LIN {X 0,Y 310.79,Z 469.746,A -85,B 0,C 180,E1 -15567.408,E2 -15567.408} C_VEL
LIN {X 0,Y 310.865,Z 470.154,A -85,B 0,C 180,E1 -15568.705,E2 -15568.705} C_VEL
LIN {X 0,Y 311.02,Z 469.974,A -85,B 0,C 180,E1 -15570,E2 -15570} C_VEL
LIN {X 0,Y 310.921,Z 469.285,A -85,B 0,C 180,E1 -15571.296,E2 -15571.296} C_VEL
LIN {X 0,Y 310.834,Z 468.094,A -85,B 0,C 180,E1 -15572.592,E2 -15572.592} C_VEL
LIN {X 0,Y 310.902,Z 466.384,A -85,B 0,C 180,E1 -15573.889,E2 -15573.889} C_VEL
LIN {X 0,Y 310.831,Z 464.037,A -85,B 0,C 180,E1 -15575.189,E2 -15575.189} C_VEL
LIN {X 0,Y 311.032,Z 459.255,A -85,B 0,C 180,E1 -15577.139,E2 -15577.139} C_VEL
LIN {X 0,Y 311.34,Z 454.023,A -85,B 0,C 180,E1 -15578.764,E2 -15578.764} C_VEL
LIN {X 0,Y 311.659,Z 448.881,A -85,B 0,C 180,E1 -15580.065,E2 -15580.065} C_VEL
LIN {X 0,Y 312.198,Z 442.687,A -85,B 0,C 180,E1 -15581.36,E2 -15581.36} C_VEL
LIN {X 0,Y 312.796,Z 436.181,A -85,B 0,C 180,E1 -15582.489,E2 -15582.489} C_VEL
LIN {X 0,Y 313.49,Z 428.304,A -85,B 0,C 180,E1 -15583.615,E2 -15583.615} C_VEL
LIN {X 0,Y 314.177,Z 420.016,A -85,B 0,C 180,E1 -15584.576,E2 -15584.576} C_VEL
LIN {X 0,Y 314.912,Z 409.522,A -85,B 0,C 180,E1 -15585.534,E2 -15585.534} C_VEL
LIN {X 0,Y 315.686,Z 397.677,A -85,B 0,C 180,E1 -15586.282,E2 -15586.282} C_VEL
LIN {X 0,Y 316.118,Z 388.576,A -85,B 0,C 180,E1 -15586.674,E2 -15586.674} C_VEL
LIN {X 0,Y 316.81,Z 345.999,A -85,B 0,C 180,E1 -15587.795,E2 -15587.795} C_VEL
LIN {X 0,Y 313.032,Z 310.136,A -85,B 0,C 180,E1 -15588.921,E2 -15588.921} C_VEL
LIN {X 0,Y 314.417,Z 295.649,A -85,B 0,C 180,E1 -15593.027,E2 -15593.027} C_VEL
LIN {X 0,Y 314.951,Z 289.674,A -85,B 0,C 180,E1 -15594.733,E2 -15594.733} C_VEL
LIN {X 0,Y 313.279,Z 279.811,A -85,B 0,C 180,E1 -15597.742,E2 -15597.742} C_VEL
LIN {X 0,Y 312.618,Z 276.356,A -85,B 0,C 180,E1 -15598.878,E2 -15598.878} C_VEL
LIN {X 0,Y 312.505,Z 276.368,A -85,B 0,C 180,E1 -15602.666,E2 -15602.666} C_VEL
LIN {X 0,Y 312.538,Z 276.365,A -85,B 0,C 180,E1 -15605.949,E2 -15605.949} C_VEL
LIN {X 0,Y 312.509,Z 276.368,A -85,B 0,C 180,E1 -15609.027,E2 -15609.027} C_VEL
LIN {X 0,Y 312.513,Z 276.366,A -85,B 0,C 180,E1 -15612.427,E2 -15612.427} C_VEL
LIN {X 0,Y 312.458,Z 276.375,A -85,B 0,C 180,E1 -15616.034,E2 -15616.034} C_VEL
LIN {X 0,Y 312.504,Z 276.37,A -85,B 0,C 180,E1 -15619.874,E2 -15619.874} C_VEL
LIN {X 0,Y 312.534,Z 276.365,A -85,B 0,C 180,E1 -15624.05,E2 -15624.05} C_VEL
LIN {X 0,Y 312.504,Z 276.371,A -85,B 0,C 180,E1 -15627.333,E2 -15627.333} C_VEL
LIN {X 0,Y 312.551,Z 276.364,A -85,B 0,C 180,E1 -15631.275,E2 -15631.275} C_VEL
LIN {X 0,Y 312.584,Z 276.358,A -85,B 0,C 180,E1 -15634.71,E2 -15634.71} C_VEL
LIN {X 0,Y 312.585,Z 276.362,A -85,B 0,C 180,E1 -15637.528,E2 -15637.528} C_VEL
LIN {X 0,Y 312.636,Z 276.356,A -85,B 0,C 180,E1 -15641.655,E2 -15641.655} C_VEL
LIN {X 0,Y 312.691,Z 276.349,A -85,B 0,C 180,E1 -15645.685,E2 -15645.685} C_VEL
LIN {X 0,Y 312.695,Z 276.349,A -85,B 0,C 180,E1 -15649.641,E2 -15649.641} C_VEL
LIN {X 0,Y 312.85,Z 276.325,A -85,B 0,C 180,E1 -15652.253,E2 -15652.253} C_VEL
LIN {X 0,Y 312.712,Z 276.341,A -85,B 0,C 180,E1 -15654.841,E2 -15654.841} C_VEL
LIN {X 0,Y 312.986,Z 276.307,A -85,B 0,C 180,E1 -15658.712,E2 -15658.712} C_VEL
LIN {X 0,Y 312.986,Z 276.31,A -85,B 0,C 180,E1 -15661.286,E2 -15661.286} C_VEL
LIN {X 0,Y 312.713,Z 276.343,A -85,B 0,C 180,E1 -15665.157,E2 -15665.157} C_VEL
LIN {X 0,Y 312.867,Z 276.327,A -85,B 0,C 180,E1 -15667.745,E2 -15667.745} C_VEL
LIN {X 0,Y 312.666,Z 276.353,A -85,B 0,C 180,E1 -15671.67,E2 -15671.67} C_VEL
LIN {X 0,Y 312.694,Z 276.344,A -85,B 0,C 180,E1 -15674.886,E2 -15674.886} C_VEL
LIN {X 0,Y 312.627,Z 276.354,A -85,B 0,C 180,E1 -15679.237,E2 -15679.237} C_VEL
LIN {X 0,Y 312.54,Z 276.363,A -85,B 0,C 180,E1 -15682.788,E2 -15682.788} C_VEL
LIN {X 0,Y 312.596,Z 276.359,A -85,B 0,C 180,E1 -15685.934,E2 -15685.934} C_VEL
LIN {X 0,Y 312.538,Z 276.368,A -85,B 0,C 180,E1 -15689.649,E2 -15689.649} C_VEL
LIN {X 0,Y 312.512,Z 276.372,A -85,B 0,C 180,E1 -15693.688,E2 -15693.688} C_VEL
LIN {X 0,Y 312.545,Z 276.365,A -85,B 0,C 180,E1 -15697.381,E2 -15697.381} C_VEL
LIN {X 0,Y 312.495,Z 276.369,A -85,B 0,C 180,E1 -15700.706,E2 -15700.706} C_VEL
LIN {X 0,Y 312.524,Z 276.366,A -85,B 0,C 180,E1 -15704.195,E2 -15704.195} C_VEL
LIN {X 0,Y 312.542,Z 276.367,A -85,B 0,C 180,E1 -15707.905,E2 -15707.905} C_VEL
LIN {X 0,Y 312.55,Z 276.366,A -85,B 0,C 180,E1 -15711.904,E2 -15711.904} C_VEL
LIN {X 0,Y 312.498,Z 276.374,A -85,B 0,C 180,E1 -15715.789,E2 -15715.789} C_VEL
LIN {X 0,Y 312.515,Z 276.366,A -85,B 0,C 180,E1 -15718.853,E2 -15718.853} C_VEL
LIN {X 0,Y 312.566,Z 276.365,A -85,B 0,C 180,E1 -15721.824,E2 -15721.824} C_VEL
LIN {X 0,Y 312.577,Z 276.358,A -85,B 0,C 180,E1 -15724.71,E2 -15724.71} C_VEL
LIN {X 0,Y 312.579,Z 276.361,A -85,B 0,C 180,E1 -15727.529,E2 -15727.529} C_VEL
LIN {X 0,Y 312.63,Z 276.356,A -85,B 0,C 180,E1 -15731.656,E2 -15731.656} C_VEL
LIN {X 0,Y 312.686,Z 276.35,A -85,B 0,C 180,E1 -15735.686,E2 -15735.686} C_VEL
LIN {X 0,Y 312.694,Z 276.348,A -85,B 0,C 180,E1 -15739.641,E2 -15739.641} C_VEL
LIN {X 0,Y 312.863,Z 276.324,A -85,B 0,C 180,E1 -15742.254,E2 -15742.254} C_VEL
LIN {X 0,Y 312.707,Z 276.342,A -85,B 0,C 180,E1 -15744.842,E2 -15744.842} C_VEL
LIN {X 0,Y 312.982,Z 276.308,A -85,B 0,C 180,E1 -15748.713,E2 -15748.713} C_VEL
LIN {X 0,Y 312.982,Z 276.309,A -85,B 0,C 180,E1 -15751.286,E2 -15751.286} C_VEL
LIN {X 0,Y 312.705,Z 276.343,A -85,B 0,C 180,E1 -15755.157,E2 -15755.157} C_VEL
LIN {X 0,Y 312.857,Z 276.328,A -85,B 0,C 180,E1 -15757.746,E2 -15757.746} C_VEL
LIN {X 0,Y 312.663,Z 276.352,A -85,B 0,C 180,E1 -15761.671,E2 -15761.671} C_VEL
LIN {X 0,Y 312.691,Z 276.344,A -85,B 0,C 180,E1 -15764.887,E2 -15764.887} C_VEL
LIN {X 0,Y 312.62,Z 276.354,A -85,B 0,C 180,E1 -15769.236,E2 -15769.236} C_VEL
LIN {X 0,Y 312.518,Z 276.366,A -85,B 0,C 180,E1 -15772.781,E2 -15772.781} C_VEL
LIN {X 0,Y 312.592,Z 276.362,A -85,B 0,C 180,E1 -15775.935,E2 -15775.935} C_VEL
LIN {X 0,Y 312.628,Z 276.487,A -85,B 0,C 180,E1 -15780.151,E2 -15780.151} C_VEL
LIN {X 0,Y 316.262,Z 290.124,A -85,B 0,C 180,E1 -15780.69,E2 -15780.69} C_VEL
LIN {X 0,Y 317.61,Z 298.066,A -85,B 0,C 180,E1 -15780.961,E2 -15780.961} C_VEL
LIN {X 0,Y 316.407,Z 353.531,A -85,B 0,C 180,E1 -15782.395,E2 -15782.395} C_VEL
LIN {X 0,Y 316.063,Z 363.172,A -85,B 0,C 180,E1 -15782.81,E2 -15782.81} C_VEL
LIN {X 0,Y 315.661,Z 373.664,A -85,B 0,C 180,E1 -15783.469,E2 -15783.469} C_VEL
LIN {X 0,Y 315.027,Z 383.974,A -85,B 0,C 180,E1 -15784.37,E2 -15784.37} C_VEL
LIN {X 0,Y 314.498,Z 392.833,A -85,B 0,C 180,E1 -15785.373,E2 -15785.373} C_VEL
LIN {X 0,Y 313.829,Z 400.58,A -85,B 0,C 180,E1 -15786.45,E2 -15786.45} C_VEL
LIN {X 0,Y 313.237,Z 406.85,A -85,B 0,C 180,E1 -15787.496,E2 -15787.496} C_VEL
LIN {X 0,Y 312.678,Z 413.25,A -85,B 0,C 180,E1 -15788.781,E2 -15788.781} C_VEL
LIN {X 0,Y 312.251,Z 418.582,A -85,B 0,C 180,E1 -15790.073,E2 -15790.073} C_VEL
LIN {X 0,Y 311.761,Z 423.009,A -85,B 0,C 180,E1 -15791.357,E2 -15791.357} C_VEL
LIN {X 0,Y 311.393,Z 427.97,A -85,B 0,C 180,E1 -15793.173,E2 -15793.173} C_VEL
LIN {X 0,Y 311.139,Z 430.66,A -85,B 0,C 180,E1 -15794.444,E2 -15794.444} C_VEL
LIN {X 0,Y 310.846,Z 433.632,A -85,B 0,C 180,E1 -15796.342,E2 -15796.342} C_VEL
LIN {X 0,Y 310.717,Z 435.486,A -85,B 0,C 180,E1 -15798.279,E2 -15798.279} C_VEL
LIN {X 0,Y 310.853,Z 436.168,A -85,B 0,C 180,E1 -15800.235,E2 -15800.235} C_VEL
LIN {X 0,Y 311.126,Z 435.457,A -85,B 0,C 180,E1 -15802.42,E2 -15802.42} C_VEL
LIN {X 0,Y 311.755,Z 432.834,A -85,B 0,C 180,E1 -15805.016,E2 -15805.016} C_VEL
LIN {X 0,Y 312.419,Z 429.501,A -85,B 0,C 180,E1 -15806.874,E2 -15806.874} C_VEL
LIN {X 0,Y 313.123,Z 425.447,A -85,B 0,C 180,E1 -15808.526,E2 -15808.526} C_VEL
LIN {X 0,Y 313.952,Z 420.392,A -85,B 0,C 180,E1 -15810.129,E2 -15810.129} C_VEL
LIN {X 0,Y 314.722,Z 415.473,A -85,B 0,C 180,E1 -15811.397,E2 -15811.397} C_VEL
LIN {X 0,Y 315.617,Z 410.145,A -85,B 0,C 180,E1 -15812.541,E2 -15812.541} C_VEL
LIN {X 0,Y 316.642,Z 402.89,A -85,B 0,C 180,E1 -15813.825,E2 -15813.825} C_VEL
LIN {X 0,Y 316.901,Z 401.141,A -85,B 0,C 180,E1 -15814.099,E2 -15814.099} C_VEL
LIN {X 0,Y 316.944,Z 396.688,A -85,B 0,C 180,E1 -15814.803,E2 -15814.803} C_VEL
LIN {X 0,Y 315.234,Z 389.246,A -85,B 0,C 180,E1 -15815.954,E2 -15815.954} C_VEL
LIN {X 0,Y 313.375,Z 381.279,A -85,B 0,C 180,E1 -15816.97,E2 -15816.97} C_VEL
LIN {X 0,Y 313.161,Z 376.007,A -85,B 0,C 180,E1 -15817.451,E2 -15817.451} C_VEL
LIN {X 0,Y 313.835,Z 365.078,A -85,B 0,C 180,E1 -15818.166,E2 -15818.166} C_VEL
LIN {X 0,Y 314.322,Z 354.986,A -85,B 0,C 180,E1 -15818.61,E2 -15818.61} C_VEL
LIN {X 0,Y 315.93,Z 301.668,A -85,B 0,C 180,E1 -15820.067,E2 -15820.067} C_VEL
LIN {X 0,Y 309.852,Z 287.044,A -85,B 0,C 180,E1 -15821.116,E2 -15821.116} C_VEL
LIN {X 0,Y 305.843,Z 278.339,A -85,B 0,C 180,E1 -15821.842,E2 -15821.842} C_VEL
LIN {X 0,Y 305.572,Z 277.239,A -85,B 0,C 180,E1 -15822.259,E2 -15822.259} C_VEL
LIN {X 0,Y 305.64,Z 277.227,A -85,B 0,C 180,E1 -15825.35,E2 -15825.35} C_VEL
LIN {X 0,Y 305.627,Z 277.228,A -85,B 0,C 180,E1 -15829.401,E2 -15829.401} C_VEL
LIN {X 0,Y 305.789,Z 277.206,A -85,B 0,C 180,E1 -15832.075,E2 -15832.075} C_VEL
LIN {X 0,Y 305.682,Z 277.217,A -85,B 0,C 180,E1 -15834.725,E2 -15834.725} C_VEL
LIN {X 0,Y 305.95,Z 277.186,A -85,B 0,C 180,E1 -15838.685,E2 -15838.685} C_VEL
LIN {X 0,Y 305.952,Z 277.181,A -85,B 0,C 180,E1 -15841.317,E2 -15841.317} C_VEL
LIN {X 0,Y 305.845,Z 277.201,A -85,B 0,C 180,E1 -15846.599,E2 -15846.599} C_VEL
LIN {X 0,Y 305.729,Z 277.211,A -85,B 0,C 180,E1 -15849.261,E2 -15849.261} C_VEL
LIN {X 0,Y 305.582,Z 277.228,A -85,B 0,C 180,E1 -15853.297,E2 -15853.297} C_VEL
LIN {X 0,Y 305.588,Z 277.225,A -85,B 0,C 180,E1 -15856.021,E2 -15856.021} C_VEL
LIN {X 0,Y 305.572,Z 277.231,A -85,B 0,C 180,E1 -15859.446,E2 -15859.446} C_VEL
LIN {X 0,Y 305.485,Z 277.243,A -85,B 0,C 180,E1 -15863.042,E2 -15863.042} C_VEL
LIN {X 0,Y 305.549,Z 277.23,A -85,B 0,C 180,E1 -15866.231,E2 -15866.231} C_VEL
LIN {X 0,Y 305.491,Z 277.234,A -85,B 0,C 180,E1 -15869.051,E2 -15869.051} C_VEL
LIN {X 0,Y 305.441,Z 277.251,A -85,B 0,C 180,E1 -15871.953,E2 -15871.953} C_VEL
LIN {X 0,Y 305.459,Z 277.249,A -85,B 0,C 180,E1 -15875.115,E2 -15875.115} C_VEL
LIN {X 0,Y 305.48,Z 277.245,A -85,B 0,C 180,E1 -15878.538,E2 -15878.538} C_VEL
LIN {X 0,Y 305.494,Z 277.245,A -85,B 0,C 180,E1 -15882.595,E2 -15882.595} C_VEL
LIN {X 0,Y 305.442,Z 277.248,A -85,B 0,C 180,E1 -15886.349,E2 -15886.349} C_VEL
LIN {X 0,Y 305.457,Z 277.249,A -85,B 0,C 180,E1 -15889.894,E2 -15889.894} C_VEL
LIN {X 0,Y 305.499,Z 277.244,A -85,B 0,C 180,E1 -15893.628,E2 -15893.628} C_VEL
LIN {X 0,Y 305.465,Z 277.248,A -85,B 0,C 180,E1 -15896.484,E2 -15896.484} C_VEL
LIN {X 0,Y 305.472,Z 277.401,A -85,B 0,C 180,E1 -15898.423,E2 -15898.423} C_VEL
LIN {X 0,Y 307.594,Z 285.931,A -85,B 0,C 180,E1 -15901.328,E2 -15901.328} C_VEL
LIN {X 0,Y 309.242,Z 294.45,A -85,B 0,C 180,E1 -15904.057,E2 -15904.057} C_VEL
LIN {X 0,Y 309.221,Z 297.943,A -85,B 0,C 180,E1 -15905.076,E2 -15905.076} C_VEL
LIN {X 0,Y 308.121,Z 306.513,A -85,B 0,C 180,E1 -15907.455,E2 -15907.455} C_VEL
LIN {X 0,Y 311.702,Z 324.802,A -85,B 0,C 180,E1 -15908.395,E2 -15908.395} C_VEL
LIN {X 0,Y 314.275,Z 342.889,A -85,B 0,C 180,E1 -15909.166,E2 -15909.166} C_VEL
LIN {X 0,Y 314.794,Z 351.131,A -85,B 0,C 180,E1 -15909.452,E2 -15909.452} C_VEL
LIN {X 0,Y 313.562,Z 387.051,A -85,B 0,C 180,E1 -15910.439,E2 -15910.439} C_VEL
LIN {X 0,Y 312.761,Z 399.292,A -85,B 0,C 180,E1 -15911.02,E2 -15911.02} C_VEL
LIN {X 0,Y 311.652,Z 409.779,A -85,B 0,C 180,E1 -15911.767,E2 -15911.767} C_VEL
LIN {X 0,Y 310.591,Z 418.26,A -85,B 0,C 180,E1 -15912.554,E2 -15912.554} C_VEL
LIN {X 0,Y 309.461,Z 426.47,A -85,B 0,C 180,E1 -15913.509,E2 -15913.509} C_VEL
LIN {X 0,Y 308.325,Z 434.313,A -85,B 0,C 180,E1 -15914.635,E2 -15914.635} C_VEL
LIN {X 0,Y 307.201,Z 440.849,A -85,B 0,C 180,E1 -15915.764,E2 -15915.764} C_VEL
LIN {X 0,Y 306.261,Z 447.117,A -85,B 0,C 180,E1 -15917.072,E2 -15917.072} C_VEL
LIN {X 0,Y 305.279,Z 453.551,A -85,B 0,C 180,E1 -15918.716,E2 -15918.716} C_VEL
LIN {X 0,Y 304.439,Z 459.551,A -85,B 0,C 180,E1 -15920.701,E2 -15920.701} C_VEL
LIN {X 0,Y 304.07,Z 462.704,A -85,B 0,C 180,E1 -15922.029,E2 -15922.029} C_VEL
LIN {X 0,Y 303.732,Z 466.505,A -85,B 0,C 180,E1 -15924.255,E2 -15924.255} C_VEL
LIN {X 0,Y 303.723,Z 468.469,A -85,B 0,C 180,E1 -15926.02,E2 -15926.02} C_VEL
LIN {X 0,Y 303.71,Z 469.371,A -85,B 0,C 180,E1 -15927.348,E2 -15927.348} C_VEL
LIN {X 0,Y 303.77,Z 469.762,A -85,B 0,C 180,E1 -15928.675,E2 -15928.675} C_VEL
LIN {X 0,Y 303.93,Z 469.549,A -85,B 0,C 180,E1 -15930,E2 -15930} C_VEL
LIN {X 0,Y 303.828,Z 468.81,A -85,B 0,C 180,E1 -15931.326,E2 -15931.326} C_VEL
LIN {X 0,Y 303.755,Z 467.568,A -85,B 0,C 180,E1 -15932.653,E2 -15932.653} C_VEL
LIN {X 0,Y 303.832,Z 465.805,A -85,B 0,C 180,E1 -15933.979,E2 -15933.979} C_VEL
LIN {X 0,Y 303.812,Z 462.107,A -85,B 0,C 180,E1 -15935.893,E2 -15935.893} C_VEL
LIN {X 0,Y 303.961,Z 458.545,A -85,B 0,C 180,E1 -15937.306,E2 -15937.306} C_VEL
LIN {X 0,Y 304.281,Z 453.238,A -85,B 0,C 180,E1 -15938.969,E2 -15938.969} C_VEL
LIN {X 0,Y 304.647,Z 448.017,A -85,B 0,C 180,E1 -15940.299,E2 -15940.299} C_VEL
LIN {X 0,Y 305.185,Z 441.723,A -85,B 0,C 180,E1 -15941.625,E2 -15941.625} C_VEL
LIN {X 0,Y 305.816,Z 435.104,A -85,B 0,C 180,E1 -15942.779,E2 -15942.779} C_VEL
LIN {X 0,Y 306.489,Z 427.078,A -85,B 0,C 180,E1 -15943.932,E2 -15943.932} C_VEL
LIN {X 0,Y 307.377,Z 417.101,A -85,B 0,C 180,E1 -15945.075,E2 -15945.075} C_VEL
LIN {X 0,Y 308.176,Z 406.544,A -85,B 0,C 180,E1 -15945.967,E2 -15945.967} C_VEL
LIN {X 0,Y 308.774,Z 396.77,A -85,B 0,C 180,E1 -15946.572,E2 -15946.572} C_VEL
LIN {X 0,Y 309.194,Z 387.415,A -85,B 0,C 180,E1 -15946.974,E2 -15946.974} C_VEL
LIN {X 0,Y 309.893,Z 346.657,A -85,B 0,C 180,E1 -15948.07,E2 -15948.07} C_VEL
LIN {X 0,Y 306.062,Z 309.72,A -85,B 0,C 180,E1 -15949.263,E2 -15949.263} C_VEL
LIN {X 0,Y 307.516,Z 295.348,A -85,B 0,C 180,E1 -15953.44,E2 -15953.44} C_VEL
LIN {X 0,Y 307.887,Z 290.114,A -85,B 0,C 180,E1 -15954.979,E2 -15954.979} C_VEL
LIN {X 0,Y 306.129,Z 280.199,A -85,B 0,C 180,E1 -15958.075,E2 -15958.075} C_VEL
LIN {X 0,Y 305.557,Z 277.236,A -85,B 0,C 180,E1 -15959.069,E2 -15959.069} C_VEL
LIN {X 0,Y 305.467,Z 277.25,A -85,B 0,C 180,E1 -15963.516,E2 -15963.516} C_VEL
LIN {X 0,Y 305.482,Z 277.242,A -85,B 0,C 180,E1 -15966.738,E2 -15966.738} C_VEL
LIN {X 0,Y 305.456,Z 277.245,A -85,B 0,C 180,E1 -15970.599,E2 -15970.599} C_VEL
LIN {X 0,Y 305.429,Z 277.253,A -85,B 0,C 180,E1 -15973.654,E2 -15973.654} C_VEL
LIN {X 0,Y 305.455,Z 277.25,A -85,B 0,C 180,E1 -15977.413,E2 -15977.413} C_VEL
LIN {X 0,Y 305.475,Z 277.248,A -85,B 0,C 180,E1 -15981.597,E2 -15981.597} C_VEL
LIN {X 0,Y 305.461,Z 277.245,A -85,B 0,C 180,E1 -15984.886,E2 -15984.886} C_VEL
LIN {X 0,Y 305.451,Z 277.246,A -85,B 0,C 180,E1 -15988.354,E2 -15988.354} C_VEL
LIN {X 0,Y 305.519,Z 277.239,A -85,B 0,C 180,E1 -15991.113,E2 -15991.113} C_VEL
LIN {X 0,Y 305.57,Z 277.233,A -85,B 0,C 180,E1 -15994.087,E2 -15994.087} C_VEL
LIN {X 0,Y 305.498,Z 277.24,A -85,B 0,C 180,E1 -15998.402,E2 -15998.402} C_VEL
LIN {X 0,Y 305.588,Z 277.231,A -85,B 0,C 180,E1 -16001.217,E2 -16001.217} C_VEL
LIN {X 0,Y 305.646,Z 277.225,A -85,B 0,C 180,E1 -16005.348,E2 -16005.348} C_VEL
LIN {X 0,Y 305.632,Z 277.227,A -85,B 0,C 180,E1 -16009.398,E2 -16009.398} C_VEL
LIN {X 0,Y 305.794,Z 277.205,A -85,B 0,C 180,E1 -16012.073,E2 -16012.073} C_VEL
LIN {X 0,Y 305.683,Z 277.217,A -85,B 0,C 180,E1 -16014.722,E2 -16014.722} C_VEL
LIN {X 0,Y 305.953,Z 277.184,A -85,B 0,C 180,E1 -16018.683,E2 -16018.683} C_VEL
LIN {X 0,Y 305.953,Z 277.186,A -85,B 0,C 180,E1 -16021.315,E2 -16021.315} C_VEL
LIN {X 0,Y 305.847,Z 277.197,A -85,B 0,C 180,E1 -16026.596,E2 -16026.596} C_VEL
LIN {X 0,Y 305.731,Z 277.213,A -85,B 0,C 180,E1 -16029.259,E2 -16029.259} C_VEL
LIN {X 0,Y 305.585,Z 277.231,A -85,B 0,C 180,E1 -16033.295,E2 -16033.295} C_VEL
LIN {X 0,Y 305.588,Z 277.231,A -85,B 0,C 180,E1 -16036.019,E2 -16036.019} C_VEL
LIN {X 0,Y 305.575,Z 277.234,A -85,B 0,C 180,E1 -16039.446,E2 -16039.446} C_VEL
LIN {X 0,Y 305.484,Z 277.242,A -85,B 0,C 180,E1 -16043.04,E2 -16043.04} C_VEL
LIN {X 0,Y 305.525,Z 277.238,A -85,B 0,C 180,E1 -16046.22,E2 -16046.22} C_VEL
LIN {X 0,Y 305.487,Z 277.242,A -85,B 0,C 180,E1 -16049.048,E2 -16049.048} C_VEL
LIN {X 0,Y 305.437,Z 277.251,A -85,B 0,C 180,E1 -16051.951,E2 -16051.951} C_VEL
LIN {X 0,Y 305.456,Z 277.246,A -85,B 0,C 180,E1 -16055.112,E2 -16055.112} C_VEL
LIN {X 0,Y 305.484,Z 277.242,A -85,B 0,C 180,E1 -16058.538,E2 -16058.538} C_VEL
LIN {X 0,Y 305.491,Z 277.241,A -85,B 0,C 180,E1 -16062.594,E2 -16062.594} C_VEL
LIN {X 0,Y 305.489,Z 277.242,A -85,B 0,C 180,E1 -16066.357,E2 -16066.357} C_VEL
LIN {X 0,Y 305.477,Z 277.247,A -85,B 0,C 180,E1 -16069.896,E2 -16069.896} C_VEL
LIN {X 0,Y 305.494,Z 277.245,A -85,B 0,C 180,E1 -16073.626,E2 -16073.626} C_VEL
LIN {X 0,Y 305.457,Z 277.246,A -85,B 0,C 180,E1 -16076.483,E2 -16076.483} C_VEL
LIN {X 0,Y 305.487,Z 277.242,A -85,B 0,C 180,E1 -16080.95,E2 -16080.95} C_VEL
LIN {X 0,Y 305.563,Z 277.234,A -85,B 0,C 180,E1 -16084.087,E2 -16084.087} C_VEL
LIN {X 0,Y 305.493,Z 277.242,A -85,B 0,C 180,E1 -16088.402,E2 -16088.402} C_VEL
LIN {X 0,Y 305.582,Z 277.23,A -85,B 0,C 180,E1 -16091.217,E2 -16091.217} C_VEL
LIN {X 0,Y 305.641,Z 277.224,A -85,B 0,C 180,E1 -16095.349,E2 -16095.349} C_VEL
LIN {X 0,Y 305.63,Z 277.226,A -85,B 0,C 180,E1 -16099.399,E2 -16099.399} C_VEL
LIN {X 0,Y 305.804,Z 277.205,A -85,B 0,C 180,E1 -16102.074,E2 -16102.074} C_VEL
LIN {X 0,Y 305.679,Z 277.218,A -85,B 0,C 180,E1 -16104.723,E2 -16104.723} C_VEL
LIN {X 0,Y 305.948,Z 277.184,A -85,B 0,C 180,E1 -16108.683,E2 -16108.683} C_VEL
LIN {X 0,Y 305.948,Z 277.185,A -85,B 0,C 180,E1 -16111.316,E2 -16111.316} C_VEL
LIN {X 0,Y 305.837,Z 277.198,A -85,B 0,C 180,E1 -16116.597,E2 -16116.597} C_VEL
LIN {X 0,Y 305.727,Z 277.212,A -85,B 0,C 180,E1 -16119.259,E2 -16119.259} C_VEL
LIN {X 0,Y 305.582,Z 277.231,A -85,B 0,C 180,E1 -16123.296,E2 -16123.296} C_VEL
LIN {X 0,Y 305.585,Z 277.233,A -85,B 0,C 180,E1 -16126.02,E2 -16126.02} C_VEL
LIN {X 0,Y 305.566,Z 277.234,A -85,B 0,C 180,E1 -16129.444,E2 -16129.444} C_VEL
LIN {X 0,Y 305.477,Z 277.243,A -85,B 0,C 180,E1 -16133.039,E2 -16133.039} C_VEL
LIN {X 0,Y 305.522,Z 277.24,A -85,B 0,C 180,E1 -16136.221,E2 -16136.221} C_VEL
LIN {X 0,Y 305.565,Z 277.237,A -85,B 0,C 180,E1 -16139.791,E2 -16139.791} C_VEL
LIN {X 0,Y 309.356,Z 290.796,A -85,B 0,C 180,E1 -16140.382,E2 -16140.382} C_VEL
LIN {X 0,Y 310.704,Z 298.29,A -85,B 0,C 180,E1 -16140.647,E2 -16140.647} C_VEL
LIN {X 0,Y 309.438,Z 354.306,A -85,B 0,C 180,E1 -16142.137,E2 -16142.137} C_VEL
LIN {X 0,Y 309.141,Z 365.224,A -85,B 0,C 180,E1 -16142.639,E2 -16142.639} C_VEL
LIN {X 0,Y 308.53,Z 376.572,A -85,B 0,C 180,E1 -16143.432,E2 -16143.432} C_VEL
LIN {X 0,Y 307.94,Z 385.711,A -85,B 0,C 180,E1 -16144.292,E2 -16144.292} C_VEL
LIN {X 0,Y 307.458,Z 393.812,A -85,B 0,C 180,E1 -16145.251,E2 -16145.251} C_VEL
LIN {X 0,Y 306.774,Z 401.469,A -85,B 0,C 180,E1 -16146.353,E2 -16146.353} C_VEL
LIN {X 0,Y 306.028,Z 409.075,A -85,B 0,C 180,E1 -16147.692,E2 -16147.692} C_VEL
LIN {X 0,Y 305.364,Z 416.54,A -85,B 0,C 180,E1 -16149.323,E2 -16149.323} C_VEL
LIN {X 0,Y 304.707,Z 423.154,A -85,B 0,C 180,E1 -16151.21,E2 -16151.21} C_VEL
LIN {X 0,Y 304.446,Z 426.533,A -85,B 0,C 180,E1 -16152.381,E2 -16152.381} C_VEL
LIN {X 0,Y 304.089,Z 430.667,A -85,B 0,C 180,E1 -16154.239,E2 -16154.239} C_VEL
LIN {X 0,Y 303.785,Z 433.584,A -85,B 0,C 180,E1 -16156.051,E2 -16156.051} C_VEL
LIN {X 0,Y 303.63,Z 435.461,A -85,B 0,C 180,E1 -16157.838,E2 -16157.838} C_VEL
LIN {X 0,Y 303.716,Z 436.438,A -85,B 0,C 180,E1 -16159.783,E2 -16159.783} C_VEL
LIN {X 0,Y 303.918,Z 436.314,A -85,B 0,C 180,E1 -16161.833,E2 -16161.833} C_VEL
LIN {X 0,Y 304.376,Z 434.864,A -85,B 0,C 180,E1 -16163.913,E2 -16163.913} C_VEL
LIN {X 0,Y 305.156,Z 431.279,A -85,B 0,C 180,E1 -16166.446,E2 -16166.446} C_VEL
LIN {X 0,Y 306.11,Z 426.596,A -85,B 0,C 180,E1 -16168.595,E2 -16168.595} C_VEL
LIN {X 0,Y 307.057,Z 421.034,A -85,B 0,C 180,E1 -16170.427,E2 -16170.427} C_VEL
LIN {X 0,Y 307.866,Z 416.322,A -85,B 0,C 180,E1 -16171.689,E2 -16171.689} C_VEL
LIN {X 0,Y 309.043,Z 409.67,A -85,B 0,C 180,E1 -16173.131,E2 -16173.131} C_VEL
LIN {X 0,Y 310.193,Z 401.975,A -85,B 0,C 180,E1 -16174.487,E2 -16174.487} C_VEL
LIN {X 0,Y 311.326,Z 393.583,A -85,B 0,C 180,E1 -16175.679,E2 -16175.679} C_VEL
LIN {X 0,Y 312.472,Z 382.935,A -85,B 0,C 180,E1 -16176.854,E2 -16176.854} C_VEL
LIN {X 0,Y 313.161,Z 376.007,A -85,B 0,C 180,E1 -16177.451,E2 -16177.451} C_VEL
LIN {X 0,Y 313.02,Z 370.58,A -85,B 0,C 180,E1 -16177.886,E2 -16177.886} C_VEL
LIN {X 0,Y 310.949,Z 361.716,A -85,B 0,C 180,E1 -16178.611,E2 -16178.611} C_VEL
LIN {X 0,Y 308.672,Z 352.653,A -85,B 0,C 180,E1 -16179.206,E2 -16179.206} C_VEL
LIN {X 0,Y 308.201,Z 346.919,A -85,B 0,C 180,E1 -16179.434,E2 -16179.434} C_VEL
LIN {X 0,Y 309.684,Z 303.662,A -85,B 0,C 180,E1 -16180.617,E2 -16180.617} C_VEL
LIN {X 0,Y 303.269,Z 288.312,A -85,B 0,C 180,E1 -16181.771,E2 -16181.771} C_VEL
LIN {X 0,Y 299.412,Z 280.754,A -85,B 0,C 180,E1 -16182.455,E2 -16182.455} C_VEL
LIN {X 0,Y 298.668,Z 278.879,A -85,B 0,C 180,E1 -16182.631,E2 -16182.631} C_VEL
LIN {X 0,Y 298.529,Z 278.114,A -85,B 0,C 180,E1 -16182.975,E2 -16182.975} C_VEL
LIN {X 0,Y 298.543,Z 278.11,A -85,B 0,C 180,E1 -16186.386,E2 -16186.386} C_VEL
LIN {X 0,Y 298.72,Z 278.09,A -85,B 0,C 180,E1 -16191.156,E2 -16191.156} C_VEL
LIN {X 0,Y 298.781,Z 278.082,A -85,B 0,C 180,E1 -16193.247,E2 -16193.247} C_VEL
LIN {X 0,Y 298.916,Z 278.061,A -85,B 0,C 180,E1 -16198.654,E2 -16198.654} C_VEL
LIN {X 0,Y 298.918,Z 278.057,A -85,B 0,C 180,E1 -16201.348,E2 -16201.348} C_VEL
LIN {X 0,Y 298.791,Z 278.078,A -85,B 0,C 180,E1 -16206.755,E2 -16206.755} C_VEL
LIN {X 0,Y 298.674,Z 278.091,A -85,B 0,C 180,E1 -16209.482,E2 -16209.482} C_VEL
LIN {X 0,Y 298.546,Z 278.106,A -85,B 0,C 180,E1 -16213.617,E2 -16213.617} C_VEL
LIN {X 0,Y 298.543,Z 278.1,A -85,B 0,C 180,E1 -16216.41,E2 -16216.41} C_VEL
LIN {X 0,Y 298.507,Z 278.111,A -85,B 0,C 180,E1 -16219.656,E2 -16219.656} C_VEL
LIN {X 0,Y 298.453,Z 278.118,A -85,B 0,C 180,E1 -16223.599,E2 -16223.599} C_VEL
LIN {X 0,Y 298.488,Z 278.113,A -85,B 0,C 180,E1 -16226.576,E2 -16226.576} C_VEL
LIN {X 0,Y 298.417,Z 278.114,A -85,B 0,C 180,E1 -16229.642,E2 -16229.642} C_VEL
LIN {X 0,Y 298.392,Z 278.121,A -85,B 0,C 180,E1 -16232.802,E2 -16232.802} C_VEL
LIN {X 0,Y 298.463,Z 278.113,A -85,B 0,C 180,E1 -16236.814,E2 -16236.814} C_VEL
LIN {X 0,Y 298.417,Z 278.121,A -85,B 0,C 180,E1 -16241.096,E2 -16241.096} C_VEL
LIN {X 0,Y 298.387,Z 278.131,A -85,B 0,C 180,E1 -16244.96,E2 -16244.96} C_VEL
LIN {X 0,Y 298.386,Z 278.127,A -85,B 0,C 180,E1 -16248.914,E2 -16248.914} C_VEL
LIN {X 0,Y 298.426,Z 278.128,A -85,B 0,C 180,E1 -16252.245,E2 -16252.245} C_VEL
LIN {X 0,Y 298.408,Z 278.128,A -85,B 0,C 180,E1 -16255.582,E2 -16255.582} C_VEL
LIN {X 0,Y 298.426,Z 278.287,A -85,B 0,C 180,E1 -16257.77,E2 -16257.77} C_VEL
LIN {X 0,Y 300.702,Z 287.389,A -85,B 0,C 180,E1 -16260.991,E2 -16260.991} C_VEL
LIN {X 0,Y 302.356,Z 295.878,A -85,B 0,C 180,E1 -16263.793,E2 -16263.793} C_VEL
LIN {X 0,Y 302.532,Z 298.325,A -85,B 0,C 180,E1 -16264.549,E2 -16264.549} C_VEL
LIN {X 0,Y 301.482,Z 306.03,A -85,B 0,C 180,E1 -16266.746,E2 -16266.746} C_VEL
LIN {X 0,Y 305.448,Z 326.004,A -85,B 0,C 180,E1 -16267.814,E2 -16267.814} C_VEL
LIN {X 0,Y 307.985,Z 344.653,A -85,B 0,C 180,E1 -16268.643,E2 -16268.643} C_VEL
LIN {X 0,Y 308.373,Z 351.988,A -85,B 0,C 180,E1 -16268.902,E2 -16268.902} C_VEL
LIN {X 0,Y 307.188,Z 386.272,A -85,B 0,C 180,E1 -16269.868,E2 -16269.868} C_VEL
LIN {X 0,Y 306.345,Z 398.258,A -85,B 0,C 180,E1 -16270.428,E2 -16270.428} C_VEL
LIN {X 0,Y 305.157,Z 408.946,A -85,B 0,C 180,E1 -16271.191,E2 -16271.191} C_VEL
LIN {X 0,Y 304.061,Z 417.502,A -85,B 0,C 180,E1 -16271.993,E2 -16271.993} C_VEL
LIN {X 0,Y 302.9,Z 425.769,A -85,B 0,C 180,E1 -16272.967,E2 -16272.967} C_VEL
LIN {X 0,Y 301.814,Z 432.633,A -85,B 0,C 180,E1 -16273.948,E2 -16273.948} C_VEL
LIN {X 0,Y 300.671,Z 439.364,A -85,B 0,C 180,E1 -16275.102,E2 -16275.102} C_VEL
LIN {X 0,Y 299.536,Z 445.789,A -85,B 0,C 180,E1 -16276.431,E2 -16276.431} C_VEL
LIN {X 0,Y 298.715,Z 451.15,A -85,B 0,C 180,E1 -16277.776,E2 -16277.776} C_VEL
LIN {X 0,Y 297.95,Z 455.644,A -85,B 0,C 180,E1 -16279.123,E2 -16279.123} C_VEL
LIN {X 0,Y 297.212,Z 460.997,A -85,B 0,C 180,E1 -16281.159,E2 -16281.159} C_VEL
LIN {X 0,Y 296.763,Z 464.973,A -85,B 0,C 180,E1 -16283.2,E2 -16283.2} C_VEL
LIN {X 0,Y 296.622,Z 466.815,A -85,B 0,C 180,E1 -16284.562,E2 -16284.562} C_VEL
LIN {X 0,Y 296.634,Z 468.151,A -85,B 0,C 180,E1 -16285.925,E2 -16285.925} C_VEL
LIN {X 0,Y 296.631,Z 468.997,A -85,B 0,C 180,E1 -16287.284,E2 -16287.284} C_VEL
LIN {X 0,Y 296.678,Z 469.356,A -85,B 0,C 180,E1 -16288.643,E2 -16288.643} C_VEL
LIN {X 0,Y 296.84,Z 469.12,A -85,B 0,C 180,E1 -16290,E2 -16290} C_VEL
LIN {X 0,Y 296.736,Z 468.321,A -85,B 0,C 180,E1 -16291.357,E2 -16291.357} C_VEL
LIN {X 0,Y 296.678,Z 467.018,A -85,B 0,C 180,E1 -16292.716,E2 -16292.716} C_VEL
LIN {X 0,Y 296.717,Z 464.023,A -85,B 0,C 180,E1 -16294.756,E2 -16294.756} C_VEL
LIN {X 0,Y 296.843,Z 459.683,A -85,B 0,C 180,E1 -16296.799,E2 -16296.799} C_VEL
LIN {X 0,Y 297.177,Z 453.599,A -85,B 0,C 180,E1 -16298.843,E2 -16298.843} C_VEL
LIN {X 0,Y 297.498,Z 448.527,A -85,B 0,C 180,E1 -16300.206,E2 -16300.206} C_VEL
LIN {X 0,Y 298.054,Z 442.416,A -85,B 0,C 180,E1 -16301.562,E2 -16301.562} C_VEL
LIN {X 0,Y 298.765,Z 434.975,A -85,B 0,C 180,E1 -16302.913,E2 -16302.913} C_VEL
LIN {X 0,Y 299.453,Z 427.001,A -85,B 0,C 180,E1 -16304.093,E2 -16304.093} C_VEL
LIN {X 0,Y 300.167,Z 418.6,A -85,B 0,C 180,E1 -16305.098,E2 -16305.098} C_VEL
LIN {X 0,Y 301.079,Z 407.91,A -85,B 0,C 180,E1 -16306.093,E2 -16306.093} C_VEL
LIN {X 0,Y 301.846,Z 396.427,A -85,B 0,C 180,E1 -16306.833,E2 -16306.833} C_VEL
LIN {X 0,Y 302.248,Z 387.103,A -85,B 0,C 180,E1 -16307.246,E2 -16307.246} C_VEL
LIN {X 0,Y 303.038,Z 347.743,A -85,B 0,C 180,E1 -16308.332,E2 -16308.332} C_VEL
LIN {X 0,Y 299.076,Z 309.407,A -85,B 0,C 180,E1 -16309.594,E2 -16309.594} C_VEL
LIN {X 0,Y 300.613,Z 295.01,A -85,B 0,C 180,E1 -16313.873,E2 -16313.873} C_VEL
LIN {X 0,Y 300.773,Z 290.486,A -85,B 0,C 180,E1 -16315.241,E2 -16315.241} C_VEL
LIN {X 0,Y 298.739,Z 279.321,A -85,B 0,C 180,E1 -16318.834,E2 -16318.834} C_VEL
LIN {X 0,Y 298.499,Z 278.117,A -85,B 0,C 180,E1 -16319.274,E2 -16319.274} C_VEL
LIN {X 0,Y 298.397,Z 278.126,A -85,B 0,C 180,E1 -16322.8,E2 -16322.8} C_VEL
LIN {X 0,Y 298.453,Z 278.118,A -85,B 0,C 180,E1 -16326.808,E2 -16326.808} C_VEL
LIN {X 0,Y 298.413,Z 278.124,A -85,B 0,C 180,E1 -16331.092,E2 -16331.092} C_VEL
LIN {X 0,Y 298.355,Z 278.131,A -85,B 0,C 180,E1 -16335.034,E2 -16335.034} C_VEL
LIN {X 0,Y 298.384,Z 278.127,A -85,B 0,C 180,E1 -16338.737,E2 -16338.737} C_VEL
LIN {X 0,Y 298.413,Z 278.123,A -85,B 0,C 180,E1 -16342.241,E2 -16342.241} C_VEL
LIN {X 0,Y 298.408,Z 278.129,A -85,B 0,C 180,E1 -16345.58,E2 -16345.58} C_VEL
LIN {X 0,Y 298.395,Z 278.125,A -85,B 0,C 180,E1 -16348.79,E2 -16348.79} C_VEL
LIN {X 0,Y 298.462,Z 278.119,A -85,B 0,C 180,E1 -16351.903,E2 -16351.903} C_VEL
LIN {X 0,Y 298.484,Z 278.115,A -85,B 0,C 180,E1 -16354.923,E2 -16354.923} C_VEL
LIN {X 0,Y 298.448,Z 278.12,A -85,B 0,C 180,E1 -16359.314,E2 -16359.314} C_VEL
LIN {X 0,Y 298.535,Z 278.109,A -85,B 0,C 180,E1 -16362.178,E2 -16362.178} C_VEL
LIN {X 0,Y 298.591,Z 278.101,A -85,B 0,C 180,E1 -16364.994,E2 -16364.994} C_VEL
LIN {X 0,Y 298.588,Z 278.102,A -85,B 0,C 180,E1 -16369.145,E2 -16369.145} C_VEL
LIN {X 0,Y 298.738,Z 278.085,A -85,B 0,C 180,E1 -16371.884,E2 -16371.884} C_VEL
LIN {X 0,Y 298.654,Z 278.092,A -85,B 0,C 180,E1 -16374.598,E2 -16374.598} C_VEL
LIN {X 0,Y 298.919,Z 278.06,A -85,B 0,C 180,E1 -16378.652,E2 -16378.652} C_VEL
LIN {X 0,Y 298.919,Z 278.063,A -85,B 0,C 180,E1 -16381.346,E2 -16381.346} C_VEL
LIN {X 0,Y 298.793,Z 278.076,A -85,B 0,C 180,E1 -16386.753,E2 -16386.753} C_VEL
LIN {X 0,Y 298.676,Z 278.094,A -85,B 0,C 180,E1 -16389.479,E2 -16389.479} C_VEL
LIN {X 0,Y 298.548,Z 278.11,A -85,B 0,C 180,E1 -16393.614,E2 -16393.614} C_VEL
LIN {X 0,Y 298.543,Z 278.107,A -85,B 0,C 180,E1 -16396.408,E2 -16396.408} C_VEL
LIN {X 0,Y 298.51,Z 278.116,A -85,B 0,C 180,E1 -16399.656,E2 -16399.656} C_VEL
LIN {X 0,Y 298.451,Z 278.122,A -85,B 0,C 180,E1 -16403.597,E2 -16403.597} C_VEL
LIN {X 0,Y 298.48,Z 278.114,A -85,B 0,C 180,E1 -16406.574,E2 -16406.574} C_VEL
LIN {X 0,Y 298.413,Z 278.127,A -85,B 0,C 180,E1 -16409.64,E2 -16409.64} C_VEL
LIN {X 0,Y 298.389,Z 278.126,A -85,B 0,C 180,E1 -16412.799,E2 -16412.799} C_VEL
LIN {X 0,Y 298.463,Z 278.116,A -85,B 0,C 180,E1 -16416.813,E2 -16416.813} C_VEL
LIN {X 0,Y 298.412,Z 278.124,A -85,B 0,C 180,E1 -16421.094,E2 -16421.094} C_VEL
LIN {X 0,Y 298.452,Z 278.119,A -85,B 0,C 180,E1 -16423.115,E2 -16423.115} C_VEL
LIN {X 0,Y 298.46,Z 278.116,A -85,B 0,C 180,E1 -16426.932,E2 -16426.932} C_VEL
LIN {X 0,Y 298.429,Z 278.121,A -85,B 0,C 180,E1 -16430.998,E2 -16430.998} C_VEL
LIN {X 0,Y 298.426,Z 278.124,A -85,B 0,C 180,E1 -16433.932,E2 -16433.932} C_VEL
LIN {X 0,Y 298.387,Z 278.129,A -85,B 0,C 180,E1 -16437.983,E2 -16437.983} C_VEL
LIN {X 0,Y 298.455,Z 278.121,A -85,B 0,C 180,E1 -16441.904,E2 -16441.904} C_VEL
LIN {X 0,Y 298.478,Z 278.115,A -85,B 0,C 180,E1 -16444.924,E2 -16444.924} C_VEL
LIN {X 0,Y 298.442,Z 278.121,A -85,B 0,C 180,E1 -16449.315,E2 -16449.315} C_VEL
LIN {X 0,Y 298.53,Z 278.11,A -85,B 0,C 180,E1 -16452.179,E2 -16452.179} C_VEL
LIN {X 0,Y 298.585,Z 278.102,A -85,B 0,C 180,E1 -16454.994,E2 -16454.994} C_VEL
LIN {X 0,Y 298.586,Z 278.102,A -85,B 0,C 180,E1 -16459.146,E2 -16459.146} C_VEL
LIN {X 0,Y 298.75,Z 278.085,A -85,B 0,C 180,E1 -16461.886,E2 -16461.886} C_VEL
LIN {X 0,Y 298.65,Z 278.094,A -85,B 0,C 180,E1 -16464.599,E2 -16464.599} C_VEL
LIN {X 0,Y 298.915,Z 278.06,A -85,B 0,C 180,E1 -16468.652,E2 -16468.652} C_VEL
LIN {X 0,Y 298.915,Z 278.062,A -85,B 0,C 180,E1 -16471.347,E2 -16471.347} C_VEL
LIN {X 0,Y 298.783,Z 278.076,A -85,B 0,C 180,E1 -16476.754,E2 -16476.754} C_VEL
LIN {X 0,Y 298.672,Z 278.093,A -85,B 0,C 180,E1 -16479.48,E2 -16479.48} C_VEL
LIN {X 0,Y 298.544,Z 278.11,A -85,B 0,C 180,E1 -16483.615,E2 -16483.615} C_VEL
LIN {X 0,Y 298.54,Z 278.108,A -85,B 0,C 180,E1 -16486.408,E2 -16486.408} C_VEL
LIN {X 0,Y 298.501,Z 278.115,A -85,B 0,C 180,E1 -16489.654,E2 -16489.654} C_VEL
LIN {X 0,Y 298.419,Z 278.125,A -85,B 0,C 180,E1 -16493.6,E2 -16493.6} C_VEL
LIN {X 0,Y 298.478,Z 278.116,A -85,B 0,C 180,E1 -16496.575,E2 -16496.575} C_VEL
LIN {X 0,Y 298.528,Z 278.131,A -85,B 0,C 180,E1 -16499.499,E2 -16499.499} C_VEL
LIN {X 0,Y 302.575,Z 292.277,A -85,B 0,C 180,E1 -16500.103,E2 -16500.103} C_VEL
LIN {X 0,Y 303.818,Z 299.911,A -85,B 0,C 180,E1 -16500.374,E2 -16500.374} C_VEL
LIN {X 0,Y 302.506,Z 354.653,A -85,B 0,C 180,E1 -16501.867,E2 -16501.867} C_VEL
LIN {X 0,Y 302.191,Z 366.027,A -85,B 0,C 180,E1 -16502.405,E2 -16502.405} C_VEL
LIN {X 0,Y 301.587,Z 376.783,A -85,B 0,C 180,E1 -16503.178,E2 -16503.178} C_VEL
LIN {X 0,Y 300.953,Z 386.213,A -85,B 0,C 180,E1 -16504.086,E2 -16504.086} C_VEL
LIN {X 0,Y 300.4,Z 394.895,A -85,B 0,C 180,E1 -16505.147,E2 -16505.147} C_VEL
LIN {X 0,Y 299.765,Z 401.644,A -85,B 0,C 180,E1 -16506.146,E2 -16506.146} C_VEL
LIN {X 0,Y 299.105,Z 408.193,A -85,B 0,C 180,E1 -16507.304,E2 -16507.304} C_VEL
LIN {X 0,Y 298.535,Z 414.281,A -85,B 0,C 180,E1 -16508.597,E2 -16508.597} C_VEL
LIN {X 0,Y 298.103,Z 419.273,A -85,B 0,C 180,E1 -16509.864,E2 -16509.864} C_VEL
LIN {X 0,Y 297.57,Z 424.271,A -85,B 0,C 180,E1 -16511.398,E2 -16511.398} C_VEL
LIN {X 0,Y 297.258,Z 428.142,A -85,B 0,C 180,E1 -16512.87,E2 -16512.87} C_VEL
LIN {X 0,Y 296.904,Z 431.97,A -85,B 0,C 180,E1 -16514.757,E2 -16514.757} C_VEL
LIN {X 0,Y 296.618,Z 434.617,A -85,B 0,C 180,E1 -16516.6,E2 -16516.6} C_VEL
LIN {X 0,Y 296.538,Z 436.252,A -85,B 0,C 180,E1 -16518.427,E2 -16518.427} C_VEL
LIN {X 0,Y 296.665,Z 436.94,A -85,B 0,C 180,E1 -16520.238,E2 -16520.238} C_VEL
LIN {X 0,Y 296.86,Z 436.725,A -85,B 0,C 180,E1 -16522.011,E2 -16522.011} C_VEL
LIN {X 0,Y 297.254,Z 435.639,A -85,B 0,C 180,E1 -16523.768,E2 -16523.768} C_VEL
LIN {X 0,Y 297.82,Z 433.452,A -85,B 0,C 180,E1 -16525.681,E2 -16525.681} C_VEL
LIN {X 0,Y 298.4,Z 430.911,A -85,B 0,C 180,E1 -16527.202,E2 -16527.202} C_VEL
LIN {X 0,Y 299.197,Z 427.173,A -85,B 0,C 180,E1 -16528.886,E2 -16528.886} C_VEL
LIN {X 0,Y 300.074,Z 422.426,A -85,B 0,C 180,E1 -16530.54,E2 -16530.54} C_VEL
LIN {X 0,Y 301.155,Z 416.454,A -85,B 0,C 180,E1 -16532.179,E2 -16532.179} C_VEL
LIN {X 0,Y 302.392,Z 409.932,A -85,B 0,C 180,E1 -16533.611,E2 -16533.611} C_VEL
LIN {X 0,Y 303.467,Z 403.025,A -85,B 0,C 180,E1 -16534.861,E2 -16534.861} C_VEL
LIN {X 0,Y 304.444,Z 396.423,A -85,B 0,C 180,E1 -16535.848,E2 -16535.848} C_VEL
LIN {X 0,Y 305.517,Z 387.505,A -85,B 0,C 180,E1 -16536.944,E2 -16536.944} C_VEL
LIN {X 0,Y 306.68,Z 376.705,A -85,B 0,C 180,E1 -16537.962,E2 -16537.962} C_VEL
LIN {X 0,Y 307.428,Z 365.215,A -85,B 0,C 180,E1 -16538.727,E2 -16538.727} C_VEL
LIN {X 0,Y 307.922,Z 355.353,A -85,B 0,C 180,E1 -16539.17,E2 -16539.17} C_VEL
LIN {X 0,Y 308.201,Z 346.919,A -85,B 0,C 180,E1 -16539.434,E2 -16539.434} C_VEL
LIN {X 0,Y 307.779,Z 341.138,A -85,B 0,C 180,E1 -16539.651,E2 -16539.651} C_VEL
LIN {X 0,Y 303.361,Z 322.574,A -85,B 0,C 180,E1 -16540.669,E2 -16540.669} C_VEL
LIN {X 0,Y 303.017,Z 316.793,A -85,B 0,C 180,E1 -16540.888,E2 -16540.888} C_VEL
LIN {X 0,Y 303.411,Z 305.521,A -85,B 0,C 180,E1 -16541.206,E2 -16541.206} C_VEL
LIN {X 0,Y 296.952,Z 290.192,A -85,B 0,C 180,E1 -16542.425,E2 -16542.425} C_VEL
LIN {X 0,Y 292.827,Z 282.311,A -85,B 0,C 180,E1 -16543.19,E2 -16543.19} C_VEL
LIN {X 0,Y 291.667,Z 279.919,A -85,B 0,C 180,E1 -16543.419,E2 -16543.419} C_VEL
LIN {X 0,Y 291.534,Z 279.215,A -85,B 0,C 180,E1 -16543.547,E2 -16543.547} C_VEL
LIN {X 0,Y 291.495,Z 278.99,A -85,B 0,C 180,E1 -16543.904,E2 -16543.904} C_VEL
LIN {X 0,Y 291.512,Z 278.986,A -85,B 0,C 180,E1 -16547.47,E2 -16547.47} C_VEL
LIN {X 0,Y 291.68,Z 278.965,A -85,B 0,C 180,E1 -16551.689,E2 -16551.689} C_VEL
LIN {X 0,Y 291.622,Z 278.969,A -85,B 0,C 180,E1 -16554.469,E2 -16554.469} C_VEL
LIN {X 0,Y 291.882,Z 278.937,A -85,B 0,C 180,E1 -16558.621,E2 -16558.621} C_VEL
LIN {X 0,Y 291.884,Z 278.933,A -85,B 0,C 180,E1 -16561.381,E2 -16561.381} C_VEL
LIN {X 0,Y 291.739,Z 278.955,A -85,B 0,C 180,E1 -16566.919,E2 -16566.919} C_VEL
LIN {X 0,Y 291.623,Z 278.969,A -85,B 0,C 180,E1 -16569.713,E2 -16569.713} C_VEL
LIN {X 0,Y 291.516,Z 278.983,A -85,B 0,C 180,E1 -16573.952,E2 -16573.952} C_VEL
LIN {X 0,Y 291.481,Z 278.979,A -85,B 0,C 180,E1 -16576.819,E2 -16576.819} C_VEL
LIN {X 0,Y 291.446,Z 278.989,A -85,B 0,C 180,E1 -16579.876,E2 -16579.876} C_VEL
LIN {X 0,Y 291.396,Z 278.994,A -85,B 0,C 180,E1 -16584.207,E2 -16584.207} C_VEL
LIN {X 0,Y 291.422,Z 278.996,A -85,B 0,C 180,E1 -16587.273,E2 -16587.273} C_VEL
LIN {X 0,Y 291.334,Z 279.001,A -85,B 0,C 180,E1 -16590.438,E2 -16590.438} C_VEL
LIN {X 0,Y 291.342,Z 278.996,A -85,B 0,C 180,E1 -16593.7,E2 -16593.7} C_VEL
LIN {X 0,Y 291.396,Z 278.992,A -85,B 0,C 180,E1 -16597.261,E2 -16597.261} C_VEL
LIN {X 0,Y 291.375,Z 278.997,A -85,B 0,C 180,E1 -16600.636,E2 -16600.636} C_VEL
LIN {X 0,Y 291.322,Z 279.006,A -85,B 0,C 180,E1 -16604.397,E2 -16604.397} C_VEL
LIN {X 0,Y 291.325,Z 279.009,A -85,B 0,C 180,E1 -16608.406,E2 -16608.406} C_VEL
LIN {X 0,Y 291.363,Z 279.003,A -85,B 0,C 180,E1 -16611.161,E2 -16611.161} C_VEL
LIN {X 0,Y 291.385,Z 279.003,A -85,B 0,C 180,E1 -16614.631,E2 -16614.631} C_VEL
LIN {X 0,Y 291.353,Z 279.023,A -85,B 0,C 180,E1 -16617.014,E2 -16617.014} C_VEL
LIN {X 0,Y 293.824,Z 288.882,A -85,B 0,C 180,E1 -16620.638,E2 -16620.638} C_VEL
LIN {X 0,Y 295.483,Z 297.333,A -85,B 0,C 180,E1 -16623.516,E2 -16623.516} C_VEL
LIN {X 0,Y 295.707,Z 299.77,A -85,B 0,C 180,E1 -16624.296,E2 -16624.296} C_VEL
LIN {X 0,Y 294.867,Z 305.698,A -85,B 0,C 180,E1 -16626.009,E2 -16626.009} C_VEL
LIN {X 0,Y 298.955,Z 325.783,A -85,B 0,C 180,E1 -16627.132,E2 -16627.132} C_VEL
LIN {X 0,Y 301.474,Z 343.492,A -85,B 0,C 180,E1 -16627.958,E2 -16627.958} C_VEL
LIN {X 0,Y 302.076,Z 351.964,A -85,B 0,C 180,E1 -16628.285,E2 -16628.285} C_VEL
LIN {X 0,Y 300.809,Z 386.302,A -85,B 0,C 180,E1 -16629.287,E2 -16629.287} C_VEL
LIN {X 0,Y 299.841,Z 398.689,A -85,B 0,C 180,E1 -16629.901,E2 -16629.901} C_VEL
LIN {X 0,Y 298.688,Z 408.37,A -85,B 0,C 180,E1 -16630.61,E2 -16630.61} C_VEL
LIN {X 0,Y 297.555,Z 416.748,A -85,B 0,C 180,E1 -16631.407,E2 -16631.407} C_VEL
LIN {X 0,Y 296.366,Z 425.072,A -85,B 0,C 180,E1 -16632.402,E2 -16632.402} C_VEL
LIN {X 0,Y 295.017,Z 433.018,A -85,B 0,C 180,E1 -16633.568,E2 -16633.568} C_VEL
LIN {X 0,Y 293.845,Z 439.622,A -85,B 0,C 180,E1 -16634.747,E2 -16634.747} C_VEL
LIN {X 0,Y 292.64,Z 445.94,A -85,B 0,C 180,E1 -16636.105,E2 -16636.105} C_VEL
LIN {X 0,Y 291.763,Z 451.207,A -85,B 0,C 180,E1 -16637.48,E2 -16637.48} C_VEL
LIN {X 0,Y 290.964,Z 455.618,A -85,B 0,C 180,E1 -16638.859,E2 -16638.859} C_VEL
LIN {X 0,Y 290.378,Z 459.3,A -85,B 0,C 180,E1 -16640.246,E2 -16640.246} C_VEL
LIN {X 0,Y 289.832,Z 463.565,A -85,B 0,C 180,E1 -16642.336,E2 -16642.336} C_VEL
LIN {X 0,Y 289.553,Z 466.471,A -85,B 0,C 180,E1 -16644.358,E2 -16644.358} C_VEL
LIN {X 0,Y 289.548,Z 467.836,A -85,B 0,C 180,E1 -16645.825,E2 -16645.825} C_VEL
LIN {X 0,Y 289.555,Z 468.625,A -85,B 0,C 180,E1 -16647.218,E2 -16647.218} C_VEL
LIN {X 0,Y 289.589,Z 468.934,A -85,B 0,C 180,E1 -16648.61,E2 -16648.61} C_VEL
LIN {X 0,Y 289.75,Z 468.688,A -85,B 0,C 180,E1 -16650,E2 -16650} C_VEL
LIN {X 0,Y 289.645,Z 467.832,A -85,B 0,C 180,E1 -16651.391,E2 -16651.391} C_VEL
LIN {X 0,Y 289.603,Z 466.469,A -85,B 0,C 180,E1 -16652.782,E2 -16652.782} C_VEL
LIN {X 0,Y 289.639,Z 463.407,A -85,B 0,C 180,E1 -16654.872,E2 -16654.872} C_VEL
LIN {X 0,Y 289.763,Z 458.959,A -85,B 0,C 180,E1 -16656.966,E2 -16656.966} C_VEL
LIN {X 0,Y 290.066,Z 453.945,A -85,B 0,C 180,E1 -16658.71,E2 -16658.71} C_VEL
LIN {X 0,Y 290.498,Z 447.583,A -85,B 0,C 180,E1 -16660.454,E2 -16660.454} C_VEL
LIN {X 0,Y 291.048,Z 441.354,A -85,B 0,C 180,E1 -16661.844,E2 -16661.844} C_VEL
LIN {X 0,Y 291.716,Z 434.815,A -85,B 0,C 180,E1 -16663.054,E2 -16663.054} C_VEL
LIN {X 0,Y 292.377,Z 428.139,A -85,B 0,C 180,E1 -16664.086,E2 -16664.086} C_VEL
LIN {X 0,Y 293.096,Z 420.061,A -85,B 0,C 180,E1 -16665.116,E2 -16665.116} C_VEL
LIN {X 0,Y 293.719,Z 411.724,A -85,B 0,C 180,E1 -16665.972,E2 -16665.972} C_VEL
LIN {X 0,Y 294.55,Z 402.197,A -85,B 0,C 180,E1 -16666.726,E2 -16666.726} C_VEL
LIN {X 0,Y 295.187,Z 390.387,A -85,B 0,C 180,E1 -16667.393,E2 -16667.393} C_VEL
LIN {X 0,Y 295.661,Z 372.303,A -85,B 0,C 180,E1 -16667.953,E2 -16667.953} C_VEL
LIN {X 0,Y 296.117,Z 348.174,A -85,B 0,C 180,E1 -16668.618,E2 -16668.618} C_VEL
LIN {X 0,Y 292.102,Z 308.934,A -85,B 0,C 180,E1 -16669.975,E2 -16669.975} C_VEL
LIN {X 0,Y 293.591,Z 295.693,A -85,B 0,C 180,E1 -16674.013,E2 -16674.013} C_VEL
LIN {X 0,Y 293.875,Z 292.562,A -85,B 0,C 180,E1 -16674.977,E2 -16674.977} C_VEL
LIN {X 0,Y 292.302,Z 283.401,A -85,B 0,C 180,E1 -16677.961,E2 -16677.961} C_VEL
LIN {X 0,Y 291.453,Z 278.995,A -85,B 0,C 180,E1 -16679.442,E2 -16679.442} C_VEL
LIN {X 0,Y 291.346,Z 279.007,A -85,B 0,C 180,E1 -16683.698,E2 -16683.698} C_VEL
LIN {X 0,Y 291.386,Z 279.001,A -85,B 0,C 180,E1 -16687.255,E2 -16687.255} C_VEL
LIN {X 0,Y 291.352,Z 279.002,A -85,B 0,C 180,E1 -16690.639,E2 -16690.639} C_VEL
LIN {X 0,Y 291.291,Z 279.01,A -85,B 0,C 180,E1 -16694.401,E2 -16694.401} C_VEL
LIN {X 0,Y 291.326,Z 279.006,A -85,B 0,C 180,E1 -16698.404,E2 -16698.404} C_VEL
LIN {X 0,Y 291.353,Z 279.004,A -85,B 0,C 180,E1 -16701.157,E2 -16701.157} C_VEL
LIN {X 0,Y 291.361,Z 279.001,A -85,B 0,C 180,E1 -16704.625,E2 -16704.625} C_VEL
LIN {X 0,Y 291.372,Z 279.002,A -85,B 0,C 180,E1 -16707.95,E2 -16707.95} C_VEL
LIN {X 0,Y 291.381,Z 279,A -85,B 0,C 180,E1 -16711.157,E2 -16711.157} C_VEL
LIN {X 0,Y 291.415,Z 278.995,A -85,B 0,C 180,E1 -16714.271,E2 -16714.271} C_VEL
LIN {X 0,Y 291.38,Z 279.001,A -85,B 0,C 180,E1 -16717.298,E2 -16717.298} C_VEL
LIN {X 0,Y 291.457,Z 278.99,A -85,B 0,C 180,E1 -16720.269,E2 -16720.269} C_VEL
LIN {X 0,Y 291.538,Z 278.979,A -85,B 0,C 180,E1 -16724.633,E2 -16724.633} C_VEL
LIN {X 0,Y 291.532,Z 278.98,A -85,B 0,C 180,E1 -16728.879,E2 -16728.879} C_VEL
LIN {X 0,Y 291.685,Z 278.966,A -85,B 0,C 180,E1 -16731.687,E2 -16731.687} C_VEL
LIN {X 0,Y 291.624,Z 278.968,A -85,B 0,C 180,E1 -16734.467,E2 -16734.467} C_VEL
LIN {X 0,Y 291.886,Z 278.936,A -85,B 0,C 180,E1 -16738.619,E2 -16738.619} C_VEL
LIN {X 0,Y 291.885,Z 278.939,A -85,B 0,C 180,E1 -16741.379,E2 -16741.379} C_VEL
LIN {X 0,Y 291.741,Z 278.954,A -85,B 0,C 180,E1 -16746.917,E2 -16746.917} C_VEL
LIN {X 0,Y 291.625,Z 278.973,A -85,B 0,C 180,E1 -16749.711,E2 -16749.711} C_VEL
LIN {X 0,Y 291.517,Z 278.985,A -85,B 0,C 180,E1 -16753.949,E2 -16753.949} C_VEL
LIN {X 0,Y 291.482,Z 278.986,A -85,B 0,C 180,E1 -16756.817,E2 -16756.817} C_VEL
LIN {X 0,Y 291.446,Z 278.993,A -85,B 0,C 180,E1 -16759.874,E2 -16759.874} C_VEL
LIN {X 0,Y 291.394,Z 278.999,A -85,B 0,C 180,E1 -16764.204,E2 -16764.204} C_VEL
LIN {X 0,Y 291.415,Z 278.996,A -85,B 0,C 180,E1 -16767.271,E2 -16767.271} C_VEL
LIN {X 0,Y 291.33,Z 279.005,A -85,B 0,C 180,E1 -16770.436,E2 -16770.436} C_VEL
LIN {X 0,Y 291.338,Z 279.01,A -85,B 0,C 180,E1 -16773.697,E2 -16773.697} C_VEL
LIN {X 0,Y 291.397,Z 278.998,A -85,B 0,C 180,E1 -16777.26,E2 -16777.26} C_VEL
LIN {X 0,Y 291.371,Z 279,A -85,B 0,C 180,E1 -16780.634,E2 -16780.634} C_VEL
LIN {X 0,Y 291.346,Z 279.003,A -85,B 0,C 180,E1 -16784.389,E2 -16784.389} C_VEL
LIN {X 0,Y 291.379,Z 278.999,A -85,B 0,C 180,E1 -16788.39,E2 -16788.39} C_VEL
LIN {X 0,Y 291.377,Z 279,A -85,B 0,C 180,E1 -16791.163,E2 -16791.163} C_VEL
LIN {X 0,Y 291.378,Z 278.998,A -85,B 0,C 180,E1 -16794.629,E2 -16794.629} C_VEL
LIN {X 0,Y 291.364,Z 279.005,A -85,B 0,C 180,E1 -16797.95,E2 -16797.95} C_VEL
LIN {X 0,Y 291.374,Z 279,A -85,B 0,C 180,E1 -16801.158,E2 -16801.158} C_VEL
LIN {X 0,Y 291.409,Z 278.996,A -85,B 0,C 180,E1 -16804.271,E2 -16804.271} C_VEL
LIN {X 0,Y 291.374,Z 279.001,A -85,B 0,C 180,E1 -16807.299,E2 -16807.299} C_VEL
LIN {X 0,Y 291.45,Z 278.991,A -85,B 0,C 180,E1 -16810.27,E2 -16810.27} C_VEL
LIN {X 0,Y 291.548,Z 278.978,A -85,B 0,C 180,E1 -16814.623,E2 -16814.623} C_VEL
LIN {X 0,Y 291.529,Z 278.98,A -85,B 0,C 180,E1 -16818.88,E2 -16818.88} C_VEL
LIN {X 0,Y 291.701,Z 278.963,A -85,B 0,C 180,E1 -16821.688,E2 -16821.688} C_VEL
LIN {X 0,Y 291.621,Z 278.97,A -85,B 0,C 180,E1 -16824.468,E2 -16824.468} C_VEL
LIN {X 0,Y 291.881,Z 278.936,A -85,B 0,C 180,E1 -16828.62,E2 -16828.62} C_VEL
LIN {X 0,Y 291.881,Z 278.938,A -85,B 0,C 180,E1 -16831.379,E2 -16831.379} C_VEL
LIN {X 0,Y 291.732,Z 278.954,A -85,B 0,C 180,E1 -16836.918,E2 -16836.918} C_VEL
LIN {X 0,Y 291.621,Z 278.973,A -85,B 0,C 180,E1 -16839.712,E2 -16839.712} C_VEL
LIN {X 0,Y 291.514,Z 278.986,A -85,B 0,C 180,E1 -16843.95,E2 -16843.95} C_VEL
LIN {X 0,Y 291.478,Z 278.987,A -85,B 0,C 180,E1 -16846.818,E2 -16846.818} C_VEL
LIN {X 0,Y 291.442,Z 278.997,A -85,B 0,C 180,E1 -16849.875,E2 -16849.875} C_VEL
LIN {X 0,Y 291.374,Z 279.002,A -85,B 0,C 180,E1 -16854.207,E2 -16854.207} C_VEL
LIN {X 0,Y 291.419,Z 278.996,A -85,B 0,C 180,E1 -16857.271,E2 -16857.271} C_VEL
LIN {X 0,Y 291.444,Z 278.995,A -85,B 0,C 180,E1 -16859.153,E2 -16859.153} C_VEL
LIN {X 0,Y 295.747,Z 293.472,A -85,B 0,C 180,E1 -16859.799,E2 -16859.799} C_VEL
LIN {X 0,Y 296.9,Z 301.122,A -85,B 0,C 180,E1 -16860.074,E2 -16860.074} C_VEL
LIN {X 0,Y 295.572,Z 355.16,A -85,B 0,C 180,E1 -16861.59,E2 -16861.59} C_VEL
LIN {X 0,Y 295.27,Z 365.325,A -85,B 0,C 180,E1 -16862.077,E2 -16862.077} C_VEL
LIN {X 0,Y 294.598,Z 377.629,A -85,B 0,C 180,E1 -16862.97,E2 -16862.97} C_VEL
LIN {X 0,Y 294.053,Z 385.71,A -85,B 0,C 180,E1 -16863.757,E2 -16863.757} C_VEL
LIN {X 0,Y 293.44,Z 394.797,A -85,B 0,C 180,E1 -16864.876,E2 -16864.876} C_VEL
LIN {X 0,Y 292.773,Z 401.793,A -85,B 0,C 180,E1 -16865.925,E2 -16865.925} C_VEL
LIN {X 0,Y 292.055,Z 408.745,A -85,B 0,C 180,E1 -16867.181,E2 -16867.181} C_VEL
LIN {X 0,Y 291.351,Z 416.222,A -85,B 0,C 180,E1 -16868.841,E2 -16868.841} C_VEL
LIN {X 0,Y 290.641,Z 423.012,A -85,B 0,C 180,E1 -16870.758,E2 -16870.758} C_VEL
LIN {X 0,Y 290.195,Z 428.196,A -85,B 0,C 180,E1 -16872.695,E2 -16872.695} C_VEL
LIN {X 0,Y 289.818,Z 432.211,A -85,B 0,C 180,E1 -16874.686,E2 -16874.686} C_VEL
LIN {X 0,Y 289.509,Z 435.109,A -85,B 0,C 180,E1 -16876.74,E2 -16876.74} C_VEL
LIN {X 0,Y 289.486,Z 436.954,A -85,B 0,C 180,E1 -16879.045,E2 -16879.045} C_VEL
LIN {X 0,Y 289.651,Z 437.364,A -85,B 0,C 180,E1 -16880.934,E2 -16880.934} C_VEL
LIN {X 0,Y 290.004,Z 436.654,A -85,B 0,C 180,E1 -16883.102,E2 -16883.102} C_VEL
LIN {X 0,Y 290.605,Z 434.679,A -85,B 0,C 180,E1 -16885.309,E2 -16885.309} C_VEL
LIN {X 0,Y 291.483,Z 431.3,A -85,B 0,C 180,E1 -16887.551,E2 -16887.551} C_VEL
LIN {X 0,Y 292.498,Z 426.41,A -85,B 0,C 180,E1 -16889.698,E2 -16889.698} C_VEL
LIN {X 0,Y 293.528,Z 421.356,A -85,B 0,C 180,E1 -16891.39,E2 -16891.39} C_VEL
LIN {X 0,Y 294.425,Z 416.906,A -85,B 0,C 180,E1 -16892.612,E2 -16892.612} C_VEL
LIN {X 0,Y 295.47,Z 411.619,A -85,B 0,C 180,E1 -16893.829,E2 -16893.829} C_VEL
LIN {X 0,Y 296.651,Z 404.783,A -85,B 0,C 180,E1 -16895.134,E2 -16895.134} C_VEL
LIN {X 0,Y 297.881,Z 396.953,A -85,B 0,C 180,E1 -16896.355,E2 -16896.355} C_VEL
LIN {X 0,Y 298.941,Z 388.719,A -85,B 0,C 180,E1 -16897.401,E2 -16897.401} C_VEL
LIN {X 0,Y 299.933,Z 379.842,A -85,B 0,C 180,E1 -16898.296,E2 -16898.296} C_VEL
LIN {X 0,Y 300.913,Z 369.349,A -85,B 0,C 180,E1 -16899.099,E2 -16899.099} C_VEL
LIN {X 0,Y 301.535,Z 357.761,A -85,B 0,C 180,E1 -16899.694,E2 -16899.694} C_VEL
LIN {X 0,Y 302.511,Z 330.169,A -85,B 0,C 180,E1 -16900.514,E2 -16900.514} C_VEL
LIN {X 0,Y 303.017,Z 316.793,A -85,B 0,C 180,E1 -16900.888,E2 -16900.888} C_VEL
LIN {X 0,Y 302.738,Z 312.974,A -85,B 0,C 180,E1 -16901.04,E2 -16901.04} C_VEL
LIN {X 0,Y 301.044,Z 307.623,A -85,B 0,C 180,E1 -16901.394,E2 -16901.394} C_VEL
LIN {X 0,Y 298.39,Z 302.804,A -85,B 0,C 180,E1 -16901.844,E2 -16901.844} C_VEL
LIN {X 0,Y 289.869,Z 290.446,A -85,B 0,C 180,E1 -16903.275,E2 -16903.275} C_VEL
LIN {X 0,Y 285.723,Z 283.077,A -85,B 0,C 180,E1 -16904.074,E2 -16904.074} C_VEL
LIN {X 0,Y 284.614,Z 280.537,A -85,B 0,C 180,E1 -16904.319,E2 -16904.319} C_VEL
LIN {X 0,Y 284.496,Z 279.86,A -85,B 0,C 180,E1 -16904.452,E2 -16904.452} C_VEL
LIN {X 0,Y 284.479,Z 279.864,A -85,B 0,C 180,E1 -16908.602,E2 -16908.602} C_VEL
LIN {X 0,Y 284.632,Z 279.845,A -85,B 0,C 180,E1 -16911.482,E2 -16911.482} C_VEL
LIN {X 0,Y 284.592,Z 279.846,A -85,B 0,C 180,E1 -16914.332,E2 -16914.332} C_VEL
LIN {X 0,Y 284.848,Z 279.813,A -85,B 0,C 180,E1 -16918.587,E2 -16918.587} C_VEL
LIN {X 0,Y 284.85,Z 279.809,A -85,B 0,C 180,E1 -16921.415,E2 -16921.415} C_VEL
LIN {X 0,Y 284.691,Z 279.832,A -85,B 0,C 180,E1 -16927.091,E2 -16927.091} C_VEL
LIN {X 0,Y 284.561,Z 279.85,A -85,B 0,C 180,E1 -16929.957,E2 -16929.957} C_VEL
LIN {X 0,Y 284.472,Z 279.862,A -85,B 0,C 180,E1 -16934.304,E2 -16934.304} C_VEL
LIN {X 0,Y 284.42,Z 279.859,A -85,B 0,C 180,E1 -16937.25,E2 -16937.25} C_VEL
LIN {X 0,Y 284.374,Z 279.866,A -85,B 0,C 180,E1 -16940.244,E2 -16940.244} C_VEL
LIN {X 0,Y 284.365,Z 279.873,A -85,B 0,C 180,E1 -16943.877,E2 -16943.877} C_VEL
LIN {X 0,Y 284.359,Z 279.876,A -85,B 0,C 180,E1 -16948.009,E2 -16948.009} C_VEL
LIN {X 0,Y 284.293,Z 279.885,A -85,B 0,C 180,E1 -16951.276,E2 -16951.276} C_VEL
LIN {X 0,Y 284.359,Z 279.877,A -85,B 0,C 180,E1 -16955.355,E2 -16955.355} C_VEL
LIN {X 0,Y 284.327,Z 279.876,A -85,B 0,C 180,E1 -16958.168,E2 -16958.168} C_VEL
LIN {X 0,Y 284.301,Z 279.883,A -85,B 0,C 180,E1 -16961.871,E2 -16961.871} C_VEL
LIN {X 0,Y 284.265,Z 279.888,A -85,B 0,C 180,E1 -16965.807,E2 -16965.807} C_VEL
LIN {X 0,Y 284.307,Z 279.885,A -85,B 0,C 180,E1 -16970.025,E2 -16970.025} C_VEL
LIN {X 0,Y 284.345,Z 279.879,A -85,B 0,C 180,E1 -16973.617,E2 -16973.617} C_VEL
LIN {X 0,Y 284.315,Z 279.975,A -85,B 0,C 180,E1 -16976.269,E2 -16976.269} C_VEL
LIN {X 0,Y 286.758,Z 289.473,A -85,B 0,C 180,E1 -16979.92,E2 -16979.92} C_VEL
LIN {X 0,Y 288.625,Z 298.82,A -85,B 0,C 180,E1 -16983.227,E2 -16983.227} C_VEL
LIN {X 0,Y 288.798,Z 301.85,A -85,B 0,C 180,E1 -16984.213,E2 -16984.213} C_VEL
LIN {X 0,Y 288.289,Z 305.365,A -85,B 0,C 180,E1 -16985.2,E2 -16985.2} C_VEL
LIN {X 0,Y 292.419,Z 324.835,A -85,B 0,C 180,E1 -16986.37,E2 -16986.37} C_VEL
LIN {X 0,Y 295.204,Z 344.074,A -85,B 0,C 180,E1 -16987.321,E2 -16987.321} C_VEL
LIN {X 0,Y 295.824,Z 352.496,A -85,B 0,C 180,E1 -16987.66,E2 -16987.66} C_VEL
LIN {X 0,Y 294.526,Z 385.698,A -85,B 0,C 180,E1 -16988.65,E2 -16988.65} C_VEL
LIN {X 0,Y 293.532,Z 397.996,A -85,B 0,C 180,E1 -16989.263,E2 -16989.263} C_VEL
LIN {X 0,Y 292.287,Z 407.918,A -85,B 0,C 180,E1 -16989.999,E2 -16989.999} C_VEL
LIN {X 0,Y 290.89,Z 417.672,A -85,B 0,C 180,E1 -16990.965,E2 -16990.965} C_VEL
LIN {X 0,Y 289.644,Z 425.731,A -85,B 0,C 180,E1 -16991.98,E2 -16991.98} C_VEL
LIN {X 0,Y 288.241,Z 433.472,A -85,B 0,C 180,E1 -16993.17,E2 -16993.17} C_VEL
LIN {X 0,Y 286.662,Z 441.646,A -85,B 0,C 180,E1 -16994.72,E2 -16994.72} C_VEL
LIN {X 0,Y 285.293,Z 448.85,A -85,B 0,C 180,E1 -16996.466,E2 -16996.466} C_VEL
LIN {X 0,Y 284.402,Z 453.607,A -85,B 0,C 180,E1 -16997.875,E2 -16997.875} C_VEL
LIN {X 0,Y 283.638,Z 457.568,A -85,B 0,C 180,E1 -16999.291,E2 -16999.291} C_VEL
LIN {X 0,Y 282.953,Z 462.173,A -85,B 0,C 180,E1 -17001.43,E2 -17001.43} C_VEL
LIN {X 0,Y 282.635,Z 464.563,A -85,B 0,C 180,E1 -17002.858,E2 -17002.858} C_VEL
LIN {X 0,Y 282.447,Z 466.513,A -85,B 0,C 180,E1 -17004.45,E2 -17004.45} C_VEL
LIN {X 0,Y 282.446,Z 467.531,A -85,B 0,C 180,E1 -17005.719,E2 -17005.719} C_VEL
LIN {X 0,Y 282.479,Z 468.256,A -85,B 0,C 180,E1 -17007.148,E2 -17007.148} C_VEL
LIN {X 0,Y 282.503,Z 468.5,A -85,B 0,C 180,E1 -17008.575,E2 -17008.575} C_VEL
LIN {X 0,Y 282.661,Z 468.237,A -85,B 0,C 180,E1 -17010,E2 -17010} C_VEL
LIN {X 0,Y 282.556,Z 467.341,A -85,B 0,C 180,E1 -17011.426,E2 -17011.426} C_VEL
LIN {X 0,Y 282.531,Z 465.918,A -85,B 0,C 180,E1 -17012.852,E2 -17012.852} C_VEL
LIN {X 0,Y 282.535,Z 462.382,A -85,B 0,C 180,E1 -17015.235,E2 -17015.235} C_VEL
LIN {X 0,Y 282.693,Z 458.21,A -85,B 0,C 180,E1 -17017.141,E2 -17017.141} C_VEL
LIN {X 0,Y 283.015,Z 453.093,A -85,B 0,C 180,E1 -17018.929,E2 -17018.929} C_VEL
LIN {X 0,Y 283.346,Z 448.075,A -85,B 0,C 180,E1 -17020.36,E2 -17020.36} C_VEL
LIN {X 0,Y 283.919,Z 442.024,A -85,B 0,C 180,E1 -17021.784,E2 -17021.784} C_VEL
LIN {X 0,Y 284.668,Z 434.655,A -85,B 0,C 180,E1 -17023.201,E2 -17023.201} C_VEL
LIN {X 0,Y 285.321,Z 428.019,A -85,B 0,C 180,E1 -17024.26,E2 -17024.26} C_VEL
LIN {X 0,Y 286.069,Z 420,A -85,B 0,C 180,E1 -17025.314,E2 -17025.314} C_VEL
LIN {X 0,Y 286.719,Z 411.745,A -85,B 0,C 180,E1 -17026.19,E2 -17026.19} C_VEL
LIN {X 0,Y 287.577,Z 402.322,A -85,B 0,C 180,E1 -17026.962,E2 -17026.962} C_VEL
LIN {X 0,Y 288.203,Z 391.499,A -85,B 0,C 180,E1 -17027.611,E2 -17027.611} C_VEL
LIN {X 0,Y 288.678,Z 376.254,A -85,B 0,C 180,E1 -17028.135,E2 -17028.135} C_VEL
LIN {X 0,Y 289.168,Z 348.418,A -85,B 0,C 180,E1 -17028.924,E2 -17028.924} C_VEL
LIN {X 0,Y 285.123,Z 308.623,A -85,B 0,C 180,E1 -17030.324,E2 -17030.324} C_VEL
LIN {X 0,Y 286.742,Z 294.854,A -85,B 0,C 180,E1 -17034.624,E2 -17034.624} C_VEL
LIN {X 0,Y 286.329,Z 289.958,A -85,B 0,C 180,E1 -17036.219,E2 -17036.219} C_VEL
LIN {X 0,Y 284.403,Z 279.873,A -85,B 0,C 180,E1 -17039.708,E2 -17039.708} C_VEL
LIN {X 0,Y 284.308,Z 279.882,A -85,B 0,C 180,E1 -17042.945,E2 -17042.945} C_VEL
LIN {X 0,Y 284.339,Z 279.876,A -85,B 0,C 180,E1 -17046.385,E2 -17046.385} C_VEL
LIN {X 0,Y 284.313,Z 279.881,A -85,B 0,C 180,E1 -17049.993,E2 -17049.993} C_VEL
LIN {X 0,Y 284.247,Z 279.888,A -85,B 0,C 180,E1 -17054.189,E2 -17054.189} C_VEL
LIN {X 0,Y 284.272,Z 279.885,A -85,B 0,C 180,E1 -17058.123,E2 -17058.123} C_VEL
LIN {X 0,Y 284.322,Z 279.878,A -85,B 0,C 180,E1 -17062.277,E2 -17062.277} C_VEL
LIN {X 0,Y 284.309,Z 279.883,A -85,B 0,C 180,E1 -17065.35,E2 -17065.35} C_VEL
LIN {X 0,Y 284.296,Z 279.881,A -85,B 0,C 180,E1 -17068.725,E2 -17068.725} C_VEL
LIN {X 0,Y 284.397,Z 279.869,A -85,B 0,C 180,E1 -17072.825,E2 -17072.825} C_VEL
LIN {X 0,Y 284.365,Z 279.873,A -85,B 0,C 180,E1 -17076.706,E2 -17076.706} C_VEL
LIN {X 0,Y 284.402,Z 279.87,A -85,B 0,C 180,E1 -17081.26,E2 -17081.26} C_VEL
LIN {X 0,Y 284.476,Z 279.859,A -85,B 0,C 180,E1 -17084.468,E2 -17084.468} C_VEL
LIN {X 0,Y 284.485,Z 279.857,A -85,B 0,C 180,E1 -17088.6,E2 -17088.6} C_VEL
LIN {X 0,Y 284.636,Z 279.843,A -85,B 0,C 180,E1 -17091.479,E2 -17091.479} C_VEL
LIN {X 0,Y 284.594,Z 279.844,A -85,B 0,C 180,E1 -17094.33,E2 -17094.33} C_VEL
LIN {X 0,Y 284.852,Z 279.812,A -85,B 0,C 180,E1 -17098.585,E2 -17098.585} C_VEL
LIN {X 0,Y 284.852,Z 279.815,A -85,B 0,C 180,E1 -17101.413,E2 -17101.413} C_VEL
LIN {X 0,Y 284.693,Z 279.833,A -85,B 0,C 180,E1 -17107.089,E2 -17107.089} C_VEL
LIN {X 0,Y 284.562,Z 279.85,A -85,B 0,C 180,E1 -17109.954,E2 -17109.954} C_VEL
LIN {X 0,Y 284.474,Z 279.86,A -85,B 0,C 180,E1 -17114.302,E2 -17114.302} C_VEL
LIN {X 0,Y 284.42,Z 279.868,A -85,B 0,C 180,E1 -17117.247,E2 -17117.247} C_VEL
LIN {X 0,Y 284.376,Z 279.871,A -85,B 0,C 180,E1 -17120.241,E2 -17120.241} C_VEL
LIN {X 0,Y 284.363,Z 279.877,A -85,B 0,C 180,E1 -17123.874,E2 -17123.874} C_VEL
LIN {X 0,Y 284.39,Z 279.871,A -85,B 0,C 180,E1 -17127.172,E2 -17127.172} C_VEL
LIN {X 0,Y 284.289,Z 279.883,A -85,B 0,C 180,E1 -17131.273,E2 -17131.273} C_VEL
LIN {X 0,Y 284.356,Z 279.876,A -85,B 0,C 180,E1 -17135.353,E2 -17135.353} C_VEL
LIN {X 0,Y 284.327,Z 279.878,A -85,B 0,C 180,E1 -17138.165,E2 -17138.165} C_VEL
LIN {X 0,Y 284.297,Z 279.885,A -85,B 0,C 180,E1 -17141.869,E2 -17141.869} C_VEL
LIN {X 0,Y 284.302,Z 279.884,A -85,B 0,C 180,E1 -17145.796,E2 -17145.796} C_VEL
LIN {X 0,Y 284.331,Z 279.879,A -85,B 0,C 180,E1 -17148.136,E2 -17148.136} C_VEL
LIN {X 0,Y 284.338,Z 279.877,A -85,B 0,C 180,E1 -17152.271,E2 -17152.271} C_VEL
LIN {X 0,Y 284.316,Z 279.88,A -85,B 0,C 180,E1 -17155.352,E2 -17155.352} C_VEL
LIN {X 0,Y 284.288,Z 279.883,A -85,B 0,C 180,E1 -17158.725,E2 -17158.725} C_VEL
LIN {X 0,Y 284.39,Z 279.869,A -85,B 0,C 180,E1 -17162.826,E2 -17162.826} C_VEL
LIN {X 0,Y 284.359,Z 279.874,A -85,B 0,C 180,E1 -17166.706,E2 -17166.706} C_VEL
LIN {X 0,Y 284.396,Z 279.869,A -85,B 0,C 180,E1 -17171.261,E2 -17171.261} C_VEL
LIN {X 0,Y 284.485,Z 279.858,A -85,B 0,C 180,E1 -17174.459,E2 -17174.459} C_VEL
LIN {X 0,Y 284.481,Z 279.858,A -85,B 0,C 180,E1 -17178.601,E2 -17178.601} C_VEL
LIN {X 0,Y 284.651,Z 279.839,A -85,B 0,C 180,E1 -17181.481,E2 -17181.481} C_VEL
LIN {X 0,Y 284.592,Z 279.846,A -85,B 0,C 180,E1 -17184.331,E2 -17184.331} C_VEL
LIN {X 0,Y 284.847,Z 279.812,A -85,B 0,C 180,E1 -17188.586,E2 -17188.586} C_VEL
LIN {X 0,Y 284.847,Z 279.814,A -85,B 0,C 180,E1 -17191.413,E2 -17191.413} C_VEL
LIN {X 0,Y 284.685,Z 279.832,A -85,B 0,C 180,E1 -17197.09,E2 -17197.09} C_VEL
LIN {X 0,Y 284.559,Z 279.853,A -85,B 0,C 180,E1 -17199.955,E2 -17199.955} C_VEL
LIN {X 0,Y 284.474,Z 279.86,A -85,B 0,C 180,E1 -17204.303,E2 -17204.303} C_VEL
LIN {X 0,Y 284.416,Z 279.867,A -85,B 0,C 180,E1 -17207.248,E2 -17207.248} C_VEL
LIN {X 0,Y 284.369,Z 279.875,A -85,B 0,C 180,E1 -17210.242,E2 -17210.242} C_VEL
LIN {X 0,Y 284.329,Z 279.878,A -85,B 0,C 180,E1 -17214.847,E2 -17214.847} C_VEL
LIN {X 0,Y 284.391,Z 279.928,A -85,B 0,C 180,E1 -17218.808,E2 -17218.808} C_VEL
LIN {X 0,Y 289.105,Z 295.563,A -85,B 0,C 180,E1 -17219.52,E2 -17219.52} C_VEL
LIN {X 0,Y 289.999,Z 301.629,A -85,B 0,C 180,E1 -17219.743,E2 -17219.743} C_VEL
LIN {X 0,Y 288.661,Z 354.958,A -85,B 0,C 180,E1 -17221.278,E2 -17221.278} C_VEL
LIN {X 0,Y 288.352,Z 365.069,A -85,B 0,C 180,E1 -17221.764,E2 -17221.764} C_VEL
LIN {X 0,Y 287.713,Z 376.823,A -85,B 0,C 180,E1 -17222.603,E2 -17222.603} C_VEL
LIN {X 0,Y 287.077,Z 386.213,A -85,B 0,C 180,E1 -17223.535,E2 -17223.535} C_VEL
LIN {X 0,Y 286.495,Z 394.424,A -85,B 0,C 180,E1 -17224.559,E2 -17224.559} C_VEL
LIN {X 0,Y 285.74,Z 402.195,A -85,B 0,C 180,E1 -17225.744,E2 -17225.744} C_VEL
LIN {X 0,Y 285.065,Z 408.673,A -85,B 0,C 180,E1 -17226.936,E2 -17226.936} C_VEL
LIN {X 0,Y 284.338,Z 415.967,A -85,B 0,C 180,E1 -17228.573,E2 -17228.573} C_VEL
LIN {X 0,Y 283.615,Z 422.945,A -85,B 0,C 180,E1 -17230.539,E2 -17230.539} C_VEL
LIN {X 0,Y 283.145,Z 428.238,A -85,B 0,C 180,E1 -17232.523,E2 -17232.523} C_VEL
LIN {X 0,Y 282.855,Z 431.518,A -85,B 0,C 180,E1 -17234.082,E2 -17234.082} C_VEL
LIN {X 0,Y 282.498,Z 434.717,A -85,B 0,C 180,E1 -17236.174,E2 -17236.174} C_VEL
LIN {X 0,Y 282.373,Z 436.783,A -85,B 0,C 180,E1 -17238.301,E2 -17238.301} C_VEL
LIN {X 0,Y 282.496,Z 437.725,A -85,B 0,C 180,E1 -17240.462,E2 -17240.462} C_VEL
LIN {X 0,Y 282.853,Z 437.476,A -85,B 0,C 180,E1 -17242.662,E2 -17242.662} C_VEL
LIN {X 0,Y 283.521,Z 435.493,A -85,B 0,C 180,E1 -17245.243,E2 -17245.243} C_VEL
LIN {X 0,Y 284.159,Z 433.117,A -85,B 0,C 180,E1 -17247.037,E2 -17247.037} C_VEL
LIN {X 0,Y 285.003,Z 429.825,A -85,B 0,C 180,E1 -17248.814,E2 -17248.814} C_VEL
LIN {X 0,Y 285.933,Z 425.611,A -85,B 0,C 180,E1 -17250.557,E2 -17250.557} C_VEL
LIN {X 0,Y 287.082,Z 420.305,A -85,B 0,C 180,E1 -17252.283,E2 -17252.283} C_VEL
LIN {X 0,Y 288.738,Z 412.539,A -85,B 0,C 180,E1 -17254.233,E2 -17254.233} C_VEL
LIN {X 0,Y 290.117,Z 405.124,A -85,B 0,C 180,E1 -17255.682,E2 -17255.682} C_VEL
LIN {X 0,Y 291.266,Z 398.144,A -85,B 0,C 180,E1 -17256.806,E2 -17256.806} C_VEL
LIN {X 0,Y 292.297,Z 390.801,A -85,B 0,C 180,E1 -17257.786,E2 -17257.786} C_VEL
LIN {X 0,Y 293.46,Z 381.229,A -85,B 0,C 180,E1 -17258.8,E2 -17258.8} C_VEL
LIN {X 0,Y 294.412,Z 371.717,A -85,B 0,C 180,E1 -17259.568,E2 -17259.568} C_VEL
LIN {X 0,Y 295.158,Z 359.79,A -85,B 0,C 180,E1 -17260.257,E2 -17260.257} C_VEL
LIN {X 0,Y 295.907,Z 339.947,A -85,B 0,C 180,E1 -17260.891,E2 -17260.891} C_VEL
LIN {X 0,Y 297.176,Z 307.279,A -85,B 0,C 180,E1 -17261.826,E2 -17261.826} C_VEL
LIN {X 0,Y 290.701,Z 292.219,A -85,B 0,C 180,E1 -17263.11,E2 -17263.11} C_VEL
LIN {X 0,Y 289.869,Z 290.446,A -85,B 0,C 180,E1 -17263.275,E2 -17263.275} C_VEL
LIN {X 0,Y 288.001,Z 287.742,A -85,B 0,C 180,E1 -17263.66,E2 -17263.66} C_VEL
LIN {X 0,Y 284.934,Z 284.704,A -85,B 0,C 180,E1 -17264.422,E2 -17264.422} C_VEL
LIN {X 0,Y 281.975,Z 282.684,A -85,B 0,C 180,E1 -17265.345,E2 -17265.345} C_VEL
LIN {X 0,Y 279.459,Z 281.45,A -85,B 0,C 180,E1 -17266.404,E2 -17266.404} C_VEL
LIN {X 0,Y 277.809,Z 280.849,A -85,B 0,C 180,E1 -17267.557,E2 -17267.557} C_VEL
LIN {X 0,Y 277.424,Z 280.74,A -85,B 0,C 180,E1 -17268.36,E2 -17268.36} C_VEL
LIN {X 0,Y 277.59,Z 280.722,A -85,B 0,C 180,E1 -17271.264,E2 -17271.264} C_VEL
LIN {X 0,Y 277.562,Z 280.722,A -85,B 0,C 180,E1 -17274.188,E2 -17274.188} C_VEL
LIN {X 0,Y 277.814,Z 280.689,A -85,B 0,C 180,E1 -17278.552,E2 -17278.552} C_VEL
LIN {X 0,Y 277.816,Z 280.685,A -85,B 0,C 180,E1 -17281.451,E2 -17281.451} C_VEL
LIN {X 0,Y 277.646,Z 280.709,A -85,B 0,C 180,E1 -17287.272,E2 -17287.272} C_VEL
LIN {X 0,Y 277.501,Z 280.731,A -85,B 0,C 180,E1 -17290.213,E2 -17290.213} C_VEL
LIN {X 0,Y 277.423,Z 280.741,A -85,B 0,C 180,E1 -17294.676,E2 -17294.676} C_VEL
LIN {X 0,Y 277.341,Z 280.748,A -85,B 0,C 180,E1 -17299.235,E2 -17299.235} C_VEL
LIN {X 0,Y 277.315,Z 280.747,A -85,B 0,C 180,E1 -17304.172,E2 -17304.172} C_VEL
LIN {X 0,Y 277.332,Z 280.751,A -85,B 0,C 180,E1 -17307.51,E2 -17307.51} C_VEL
LIN {X 0,Y 277.269,Z 280.753,A -85,B 0,C 180,E1 -17310.483,E2 -17310.483} C_VEL
LIN {X 0,Y 277.251,Z 280.752,A -85,B 0,C 180,E1 -17313.896,E2 -17313.896} C_VEL
LIN {X 0,Y 277.283,Z 280.75,A -85,B 0,C 180,E1 -17317.468,E2 -17317.468} C_VEL
LIN {X 0,Y 277.239,Z 280.759,A -85,B 0,C 180,E1 -17321.232,E2 -17321.232} C_VEL
LIN {X 0,Y 277.219,Z 280.767,A -85,B 0,C 180,E1 -17325.224,E2 -17325.224} C_VEL
LIN {X 0,Y 277.222,Z 280.764,A -85,B 0,C 180,E1 -17329.514,E2 -17329.514} C_VEL
LIN {X 0,Y 277.276,Z 280.763,A -85,B 0,C 180,E1 -17332.533,E2 -17332.533} C_VEL
LIN {X 0,Y 277.293,Z 280.899,A -85,B 0,C 180,E1 -17335.453,E2 -17335.453} C_VEL
LIN {X 0,Y 279.634,Z 289.994,A -85,B 0,C 180,E1 -17339.115,E2 -17339.115} C_VEL
LIN {X 0,Y 281.569,Z 299.152,A -85,B 0,C 180,E1 -17342.5,E2 -17342.5} C_VEL
LIN {X 0,Y 282.067,Z 302.797,A -85,B 0,C 180,E1 -17343.765,E2 -17343.765} C_VEL
LIN {X 0,Y 281.801,Z 304.586,A -85,B 0,C 180,E1 -17344.321,E2 -17344.321} C_VEL
LIN {X 0,Y 286.153,Z 325.221,A -85,B 0,C 180,E1 -17345.632,E2 -17345.632} C_VEL
LIN {X 0,Y 288.96,Z 344.412,A -85,B 0,C 180,E1 -17346.631,E2 -17346.631} C_VEL
LIN {X 0,Y 289.591,Z 353.621,A -85,B 0,C 180,E1 -17347.018,E2 -17347.018} C_VEL
LIN {X 0,Y 288.23,Z 385.053,A -85,B 0,C 180,E1 -17347.978,E2 -17347.978} C_VEL
LIN {X 0,Y 287.303,Z 396.58,A -85,B 0,C 180,E1 -17348.547,E2 -17348.547} C_VEL
LIN {X 0,Y 285.967,Z 407.226,A -85,B 0,C 180,E1 -17349.34,E2 -17349.34} C_VEL
LIN {X 0,Y 284.48,Z 417.109,A -85,B 0,C 180,E1 -17350.331,E2 -17350.331} C_VEL
LIN {X 0,Y 283.158,Z 425.196,A -85,B 0,C 180,E1 -17351.365,E2 -17351.365} C_VEL
LIN {X 0,Y 281.713,Z 432.957,A -85,B 0,C 180,E1 -17352.581,E2 -17352.581} C_VEL
LIN {X 0,Y 279.848,Z 441.97,A -85,B 0,C 180,E1 -17354.338,E2 -17354.338} C_VEL
LIN {X 0,Y 278.38,Z 448.976,A -85,B 0,C 180,E1 -17356.124,E2 -17356.124} C_VEL
LIN {X 0,Y 277.472,Z 453.624,A -85,B 0,C 180,E1 -17357.568,E2 -17357.568} C_VEL
LIN {X 0,Y 276.657,Z 457.52,A -85,B 0,C 180,E1 -17359.017,E2 -17359.017} C_VEL
LIN {X 0,Y 275.926,Z 462.004,A -85,B 0,C 180,E1 -17361.21,E2 -17361.21} C_VEL
LIN {X 0,Y 275.587,Z 464.333,A -85,B 0,C 180,E1 -17362.675,E2 -17362.675} C_VEL
LIN {X 0,Y 275.358,Z 466.413,A -85,B 0,C 180,E1 -17364.511,E2 -17364.511} C_VEL
LIN {X 0,Y 275.405,Z 467.887,A -85,B 0,C 180,E1 -17367.075,E2 -17367.075} C_VEL
LIN {X 0,Y 275.42,Z 468.063,A -85,B 0,C 180,E1 -17368.538,E2 -17368.538} C_VEL
LIN {X 0,Y 275.573,Z 467.758,A -85,B 0,C 180,E1 -17370,E2 -17370} C_VEL
LIN {X 0,Y 275.471,Z 466.837,A -85,B 0,C 180,E1 -17371.462,E2 -17371.462} C_VEL
LIN {X 0,Y 275.483,Z 464.463,A -85,B 0,C 180,E1 -17373.657,E2 -17373.657} C_VEL
LIN {X 0,Y 275.533,Z 460.677,A -85,B 0,C 180,E1 -17375.856,E2 -17375.856} C_VEL
LIN {X 0,Y 275.75,Z 455.445,A -85,B 0,C 180,E1 -17378.058,E2 -17378.058} C_VEL
LIN {X 0,Y 276.133,Z 449.786,A -85,B 0,C 180,E1 -17379.893,E2 -17379.893} C_VEL
LIN {X 0,Y 276.795,Z 442.616,A -85,B 0,C 180,E1 -17381.72,E2 -17381.72} C_VEL
LIN {X 0,Y 277.593,Z 434.401,A -85,B 0,C 180,E1 -17383.357,E2 -17383.357} C_VEL
LIN {X 0,Y 278.275,Z 427.797,A -85,B 0,C 180,E1 -17384.442,E2 -17384.442} C_VEL
LIN {X 0,Y 279.045,Z 419.82,A -85,B 0,C 180,E1 -17385.522,E2 -17385.522} C_VEL
LIN {X 0,Y 279.724,Z 411.622,A -85,B 0,C 180,E1 -17386.419,E2 -17386.419} C_VEL
LIN {X 0,Y 280.609,Z 402.296,A -85,B 0,C 180,E1 -17387.209,E2 -17387.209} C_VEL
LIN {X 0,Y 281.156,Z 392.778,A -85,B 0,C 180,E1 -17387.809,E2 -17387.809} C_VEL
LIN {X 0,Y 281.639,Z 380.162,A -85,B 0,C 180,E1 -17388.317,E2 -17388.317} C_VEL
LIN {X 0,Y 282.197,Z 348.086,A -85,B 0,C 180,E1 -17389.256,E2 -17389.256} C_VEL
LIN {X 0,Y 278.178,Z 308.195,A -85,B 0,C 180,E1 -17390.714,E2 -17390.714} C_VEL
LIN {X 0,Y 279.755,Z 295.242,A -85,B 0,C 180,E1 -17394.871,E2 -17394.871} C_VEL
LIN {X 0,Y 279.167,Z 290.273,A -85,B 0,C 180,E1 -17396.542,E2 -17396.542} C_VEL
LIN {X 0,Y 277.334,Z 280.752,A -85,B 0,C 180,E1 -17399.927,E2 -17399.927} C_VEL
LIN {X 0,Y 277.249,Z 280.761,A -85,B 0,C 180,E1 -17403.895,E2 -17403.895} C_VEL
LIN {X 0,Y 277.276,Z 280.76,A -85,B 0,C 180,E1 -17407.467,E2 -17407.467} C_VEL
LIN {X 0,Y 277.222,Z 280.765,A -85,B 0,C 180,E1 -17411.234,E2 -17411.234} C_VEL
LIN {X 0,Y 277.202,Z 280.767,A -85,B 0,C 180,E1 -17415.226,E2 -17415.226} C_VEL
LIN {X 0,Y 277.223,Z 280.767,A -85,B 0,C 180,E1 -17419.511,E2 -17419.511} C_VEL
LIN {X 0,Y 277.267,Z 280.756,A -85,B 0,C 180,E1 -17422.53,E2 -17422.53} C_VEL
LIN {X 0,Y 277.247,Z 280.761,A -85,B 0,C 180,E1 -17426.103,E2 -17426.103} C_VEL
LIN {X 0,Y 277.261,Z 280.762,A -85,B 0,C 180,E1 -17429.537,E2 -17429.537} C_VEL
LIN {X 0,Y 277.358,Z 280.746,A -85,B 0,C 180,E1 -17432.863,E2 -17432.863} C_VEL
LIN {X 0,Y 277.327,Z 280.751,A -85,B 0,C 180,E1 -17436.078,E2 -17436.078} C_VEL
LIN {X 0,Y 277.343,Z 280.747,A -85,B 0,C 180,E1 -17440.765,E2 -17440.765} C_VEL
LIN {X 0,Y 277.426,Z 280.74,A -85,B 0,C 180,E1 -17445.324,E2 -17445.324} C_VEL
LIN {X 0,Y 277.459,Z 280.737,A -85,B 0,C 180,E1 -17449.786,E2 -17449.786} C_VEL
LIN {X 0,Y 277.638,Z 280.711,A -85,B 0,C 180,E1 -17452.728,E2 -17452.728} C_VEL
LIN {X 0,Y 277.818,Z 280.689,A -85,B 0,C 180,E1 -17458.549,E2 -17458.549} C_VEL
LIN {X 0,Y 277.818,Z 280.692,A -85,B 0,C 180,E1 -17461.448,E2 -17461.448} C_VEL
LIN {X 0,Y 277.648,Z 280.711,A -85,B 0,C 180,E1 -17467.27,E2 -17467.27} C_VEL
LIN {X 0,Y 277.503,Z 280.728,A -85,B 0,C 180,E1 -17470.21,E2 -17470.21} C_VEL
LIN {X 0,Y 277.424,Z 280.737,A -85,B 0,C 180,E1 -17474.673,E2 -17474.673} C_VEL
LIN {X 0,Y 277.341,Z 280.749,A -85,B 0,C 180,E1 -17479.233,E2 -17479.233} C_VEL
LIN {X 0,Y 277.323,Z 280.753,A -85,B 0,C 180,E1 -17483.919,E2 -17483.919} C_VEL
LIN {X 0,Y 277.318,Z 280.754,A -85,B 0,C 180,E1 -17487.504,E2 -17487.504} C_VEL
LIN {X 0,Y 277.266,Z 280.757,A -85,B 0,C 180,E1 -17490.48,E2 -17490.48} C_VEL
LIN {X 0,Y 277.248,Z 280.763,A -85,B 0,C 180,E1 -17493.894,E2 -17493.894} C_VEL
LIN {X 0,Y 277.283,Z 280.757,A -85,B 0,C 180,E1 -17497.465,E2 -17497.465} C_VEL
LIN {X 0,Y 277.234,Z 280.762,A -85,B 0,C 180,E1 -17501.23,E2 -17501.23} C_VEL
LIN {X 0,Y 277.244,Z 280.761,A -85,B 0,C 180,E1 -17505.215,E2 -17505.215} C_VEL
LIN {X 0,Y 277.288,Z 280.757,A -85,B 0,C 180,E1 -17509.494,E2 -17509.494} C_VEL
LIN {X 0,Y 277.283,Z 280.755,A -85,B 0,C 180,E1 -17512.534,E2 -17512.534} C_VEL
LIN {X 0,Y 277.247,Z 280.761,A -85,B 0,C 180,E1 -17516.105,E2 -17516.105} C_VEL
LIN {X 0,Y 277.254,Z 280.762,A -85,B 0,C 180,E1 -17519.538,E2 -17519.538} C_VEL
LIN {X 0,Y 277.351,Z 280.745,A -85,B 0,C 180,E1 -17522.864,E2 -17522.864} C_VEL
LIN {X 0,Y 277.321,Z 280.753,A -85,B 0,C 180,E1 -17526.079,E2 -17526.079} C_VEL
LIN {X 0,Y 277.337,Z 280.747,A -85,B 0,C 180,E1 -17530.766,E2 -17530.766} C_VEL
LIN {X 0,Y 277.427,Z 280.739,A -85,B 0,C 180,E1 -17535.325,E2 -17535.325} C_VEL
LIN {X 0,Y 277.499,Z 280.732,A -85,B 0,C 180,E1 -17539.788,E2 -17539.788} C_VEL
LIN {X 0,Y 277.645,Z 280.71,A -85,B 0,C 180,E1 -17542.729,E2 -17542.729} C_VEL
LIN {X 0,Y 277.813,Z 280.688,A -85,B 0,C 180,E1 -17548.55,E2 -17548.55} C_VEL
LIN {X 0,Y 277.813,Z 280.691,A -85,B 0,C 180,E1 -17551.449,E2 -17551.449} C_VEL
LIN {X 0,Y 277.64,Z 280.71,A -85,B 0,C 180,E1 -17557.271,E2 -17557.271} C_VEL
LIN {X 0,Y 277.499,Z 280.73,A -85,B 0,C 180,E1 -17560.211,E2 -17560.211} C_VEL
LIN {X 0,Y 277.426,Z 280.737,A -85,B 0,C 180,E1 -17564.674,E2 -17564.674} C_VEL
LIN {X 0,Y 277.336,Z 280.749,A -85,B 0,C 180,E1 -17569.234,E2 -17569.234} C_VEL
LIN {X 0,Y 277.283,Z 280.758,A -85,B 0,C 180,E1 -17574.158,E2 -17574.158} C_VEL
LIN {X 0,Y 277.344,Z 280.749,A -85,B 0,C 180,E1 -17578.439,E2 -17578.439} C_VEL
LIN {X 0,Y 282.346,Z 297.124,A -85,B 0,C 180,E1 -17579.224,E2 -17579.224} C_VEL
LIN {X 0,Y 283.084,Z 302.456,A -85,B 0,C 180,E1 -17579.423,E2 -17579.423} C_VEL
LIN {X 0,Y 281.718,Z 355.427,A -85,B 0,C 180,E1 -17580.991,E2 -17580.991} C_VEL
LIN {X 0,Y 281.407,Z 365.665,A -85,B 0,C 180,E1 -17581.5,E2 -17581.5} C_VEL
LIN {X 0,Y 280.724,Z 377.637,A -85,B 0,C 180,E1 -17582.388,E2 -17582.388} C_VEL
LIN {X 0,Y 280.083,Z 386.572,A -85,B 0,C 180,E1 -17583.298,E2 -17583.298} C_VEL
LIN {X 0,Y 279.447,Z 395.362,A -85,B 0,C 180,E1 -17584.431,E2 -17584.431} C_VEL
LIN {X 0,Y 278.814,Z 401.814,A -85,B 0,C 180,E1 -17585.432,E2 -17585.432} C_VEL
LIN {X 0,Y 278.078,Z 408.664,A -85,B 0,C 180,E1 -17586.703,E2 -17586.703} C_VEL
LIN {X 0,Y 277.361,Z 415.448,A -85,B 0,C 180,E1 -17588.235,E2 -17588.235} C_VEL
LIN {X 0,Y 276.822,Z 421.261,A -85,B 0,C 180,E1 -17589.843,E2 -17589.843} C_VEL
LIN {X 0,Y 276.191,Z 427.244,A -85,B 0,C 180,E1 -17591.908,E2 -17591.908} C_VEL
LIN {X 0,Y 275.872,Z 430.687,A -85,B 0,C 180,E1 -17593.458,E2 -17593.458} C_VEL
LIN {X 0,Y 275.487,Z 434.32,A -85,B 0,C 180,E1 -17595.585,E2 -17595.585} C_VEL
LIN {X 0,Y 275.279,Z 437.175,A -85,B 0,C 180,E1 -17598.412,E2 -17598.412} C_VEL
LIN {X 0,Y 275.414,Z 438.053,A -85,B 0,C 180,E1 -17600.363,E2 -17600.363} C_VEL
LIN {X 0,Y 275.674,Z 438.027,A -85,B 0,C 180,E1 -17602.278,E2 -17602.278} C_VEL
LIN {X 0,Y 276.196,Z 436.928,A -85,B 0,C 180,E1 -17604.512,E2 -17604.512} C_VEL
LIN {X 0,Y 277.004,Z 434.384,A -85,B 0,C 180,E1 -17606.849,E2 -17606.849} C_VEL
LIN {X 0,Y 278.132,Z 430.264,A -85,B 0,C 180,E1 -17609.216,E2 -17609.216} C_VEL
LIN {X 0,Y 279.145,Z 426.027,A -85,B 0,C 180,E1 -17611.012,E2 -17611.012} C_VEL
LIN {X 0,Y 280.424,Z 420.571,A -85,B 0,C 180,E1 -17612.82,E2 -17612.82} C_VEL
LIN {X 0,Y 282.1,Z 413.126,A -85,B 0,C 180,E1 -17614.729,E2 -17614.729} C_VEL
LIN {X 0,Y 283.515,Z 405.997,A -85,B 0,C 180,E1 -17616.163,E2 -17616.163} C_VEL
LIN {X 0,Y 284.945,Z 397.622,A -85,B 0,C 180,E1 -17617.525,E2 -17617.525} C_VEL
LIN {X 0,Y 286.036,Z 390.116,A -85,B 0,C 180,E1 -17618.519,E2 -17618.519} C_VEL
LIN {X 0,Y 287.176,Z 381.259,A -85,B 0,C 180,E1 -17619.46,E2 -17619.46} C_VEL
LIN {X 0,Y 288.291,Z 370.603,A -85,B 0,C 180,E1 -17620.324,E2 -17620.324} C_VEL
LIN {X 0,Y 288.984,Z 359.02,A -85,B 0,C 180,E1 -17620.962,E2 -17620.962} C_VEL
LIN {X 0,Y 290.007,Z 333.061,A -85,B 0,C 180,E1 -17621.785,E2 -17621.785} C_VEL
LIN {X 0,Y 290.928,Z 308.952,A -85,B 0,C 180,E1 -17622.505,E2 -17622.505} C_VEL
LIN {X 0,Y 284.728,Z 294.617,A -85,B 0,C 180,E1 -17623.787,E2 -17623.787} C_VEL
LIN {X 0,Y 278.977,Z 284.358,A -85,B 0,C 180,E1 -17624.971,E2 -17624.971} C_VEL
LIN {X 0,Y 277.568,Z 281.54,A -85,B 0,C 180,E1 -17625.283,E2 -17625.283} C_VEL
LIN {X 0,Y 277.441,Z 280.74,A -85,B 0,C 180,E1 -17625.375,E2 -17625.375} C_VEL
LIN {X 0,Y 277.424,Z 280.74,A -85,B 0,C 180,E1 -17628.36,E2 -17628.36} C_VEL
LIN {X 0,Y 276.753,Z 280.825,A -85,B 0,C 180,E1 -17629.574,E2 -17629.574} C_VEL
LIN {X 0,Y 273.976,Z 281.171,A -85,B 0,C 180,E1 -17631.555,E2 -17631.555} C_VEL
LIN {X 0,Y 271.608,Z 281.466,A -85,B 0,C 180,E1 -17633.164,E2 -17633.164} C_VEL
LIN {X 0,Y 270.554,Z 281.594,A -85,B 0,C 180,E1 -17634.409,E2 -17634.409} C_VEL
LIN {X 0,Y 270.448,Z 281.605,A -85,B 0,C 180,E1 -17634.831,E2 -17634.831} C_VEL
LIN {X 0,Y 270.78,Z 281.564,A -85,B 0,C 180,E1 -17638.514,E2 -17638.514} C_VEL
LIN {X 0,Y 270.781,Z 281.562,A -85,B 0,C 180,E1 -17641.488,E2 -17641.488} C_VEL
LIN {X 0,Y 270.605,Z 281.585,A -85,B 0,C 180,E1 -17647.463,E2 -17647.463} C_VEL
LIN {X 0,Y 270.436,Z 281.612,A -85,B 0,C 180,E1 -17650.482,E2 -17650.482} C_VEL
LIN {X 0,Y 270.391,Z 281.615,A -85,B 0,C 180,E1 -17655.066,E2 -17655.066} C_VEL
LIN {X 0,Y 270.297,Z 281.623,A -85,B 0,C 180,E1 -17659.757,E2 -17659.757} C_VEL
LIN {X 0,Y 270.271,Z 281.621,A -85,B 0,C 180,E1 -17664.587,E2 -17664.587} C_VEL
LIN {X 0,Y 270.272,Z 281.631,A -85,B 0,C 180,E1 -17667.91,E2 -17667.91} C_VEL
LIN {X 0,Y 270.182,Z 281.643,A -85,B 0,C 180,E1 -17671.35,E2 -17671.35} C_VEL
LIN {X 0,Y 270.212,Z 281.638,A -85,B 0,C 180,E1 -17674.905,E2 -17674.905} C_VEL
LIN {X 0,Y 270.221,Z 281.639,A -85,B 0,C 180,E1 -17678.718,E2 -17678.718} C_VEL
LIN {X 0,Y 270.194,Z 281.642,A -85,B 0,C 180,E1 -17682.555,E2 -17682.555} C_VEL
LIN {X 0,Y 270.171,Z 281.64,A -85,B 0,C 180,E1 -17686.751,E2 -17686.751} C_VEL
LIN {X 0,Y 270.198,Z 281.64,A -85,B 0,C 180,E1 -17691.291,E2 -17691.291} C_VEL
LIN {X 0,Y 270.301,Z 281.779,A -85,B 0,C 180,E1 -17694.541,E2 -17694.541} C_VEL
LIN {X 0,Y 272.575,Z 290.699,A -85,B 0,C 180,E1 -17698.307,E2 -17698.307} C_VEL
LIN {X 0,Y 274.304,Z 298.331,A -85,B 0,C 180,E1 -17701.29,E2 -17701.29} C_VEL
LIN {X 0,Y 275.272,Z 304.211,A -85,B 0,C 180,E1 -17703.396,E2 -17703.396} C_VEL
LIN {X 0,Y 279.136,Z 321.474,A -85,B 0,C 180,E1 -17704.593,E2 -17704.593} C_VEL
LIN {X 0,Y 281.703,Z 336.789,A -85,B 0,C 180,E1 -17705.485,E2 -17705.485} C_VEL
LIN {X 0,Y 283.308,Z 350.654,A -85,B 0,C 180,E1 -17706.172,E2 -17706.172} C_VEL
LIN {X 0,Y 283.305,Z 358.639,A -85,B 0,C 180,E1 -17706.451,E2 -17706.451} C_VEL
LIN {X 0,Y 282.054,Z 384.857,A -85,B 0,C 180,E1 -17707.276,E2 -17707.276} C_VEL
LIN {X 0,Y 281.067,Z 396.398,A -85,B 0,C 180,E1 -17707.867,E2 -17707.867} C_VEL
LIN {X 0,Y 279.714,Z 406.531,A -85,B 0,C 180,E1 -17708.635,E2 -17708.635} C_VEL
LIN {X 0,Y 278.089,Z 416.642,A -85,B 0,C 180,E1 -17709.667,E2 -17709.667} C_VEL
LIN {X 0,Y 276.714,Z 424.698,A -85,B 0,C 180,E1 -17710.721,E2 -17710.721} C_VEL
LIN {X 0,Y 275.163,Z 432.447,A -85,B 0,C 180,E1 -17711.96,E2 -17711.96} C_VEL
LIN {X 0,Y 273.425,Z 440.66,A -85,B 0,C 180,E1 -17713.577,E2 -17713.577} C_VEL
LIN {X 0,Y 271.761,Z 447.904,A -85,B 0,C 180,E1 -17715.396,E2 -17715.396} C_VEL
LIN {X 0,Y 270.552,Z 453.661,A -85,B 0,C 180,E1 -17717.245,E2 -17717.245} C_VEL
LIN {X 0,Y 269.345,Z 459.064,A -85,B 0,C 180,E1 -17719.476,E2 -17719.476} C_VEL
LIN {X 0,Y 268.888,Z 461.867,A -85,B 0,C 180,E1 -17720.978,E2 -17720.978} C_VEL
LIN {X 0,Y 268.53,Z 464.111,A -85,B 0,C 180,E1 -17722.481,E2 -17722.481} C_VEL
LIN {X 0,Y 268.264,Z 466.273,A -85,B 0,C 180,E1 -17724.586,E2 -17724.586} C_VEL
LIN {X 0,Y 268.33,Z 467.521,A -85,B 0,C 180,E1 -17726.998,E2 -17726.998} C_VEL
LIN {X 0,Y 268.339,Z 467.628,A -85,B 0,C 180,E1 -17728.5,E2 -17728.5} C_VEL
LIN {X 0,Y 268.487,Z 467.257,A -85,B 0,C 180,E1 -17730,E2 -17730} C_VEL
LIN {X 0,Y 268.388,Z 466.321,A -85,B 0,C 180,E1 -17731.501,E2 -17731.501} C_VEL
LIN {X 0,Y 268.422,Z 463.816,A -85,B 0,C 180,E1 -17733.753,E2 -17733.753} C_VEL
LIN {X 0,Y 268.436,Z 460.395,A -85,B 0,C 180,E1 -17735.789,E2 -17735.789} C_VEL
LIN {X 0,Y 268.587,Z 456.569,A -85,B 0,C 180,E1 -17737.518,E2 -17737.518} C_VEL
LIN {X 0,Y 268.854,Z 452.453,A -85,B 0,C 180,E1 -17739.024,E2 -17739.024} C_VEL
LIN {X 0,Y 269.223,Z 447.468,A -85,B 0,C 180,E1 -17740.529,E2 -17740.529} C_VEL
LIN {X 0,Y 269.785,Z 441.446,A -85,B 0,C 180,E1 -17742.029,E2 -17742.029} C_VEL
LIN {X 0,Y 270.54,Z 434.113,A -85,B 0,C 180,E1 -17743.521,E2 -17743.521} C_VEL
LIN {X 0,Y 271.239,Z 427.528,A -85,B 0,C 180,E1 -17744.633,E2 -17744.633} C_VEL
LIN {X 0,Y 272.027,Z 419.575,A -85,B 0,C 180,E1 -17745.74,E2 -17745.74} C_VEL
LIN {X 0,Y 272.733,Z 411.414,A -85,B 0,C 180,E1 -17746.659,E2 -17746.659} C_VEL
LIN {X 0,Y 273.631,Z 402.138,A -85,B 0,C 180,E1 -17747.469,E2 -17747.469} C_VEL
LIN {X 0,Y 274.226,Z 392.502,A -85,B 0,C 180,E1 -17748.095,E2 -17748.095} C_VEL
LIN {X 0,Y 274.727,Z 379.626,A -85,B 0,C 180,E1 -17748.627,E2 -17748.627} C_VEL
LIN {X 0,Y 275.313,Z 349.154,A -85,B 0,C 180,E1 -17749.543,E2 -17749.543} C_VEL
LIN {X 0,Y 271.193,Z 307.943,A -85,B 0,C 180,E1 -17751.064,E2 -17751.064} C_VEL
LIN {X 0,Y 272.71,Z 296.132,A -85,B 0,C 180,E1 -17754.948,E2 -17754.948} C_VEL
LIN {X 0,Y 272.239,Z 291.786,A -85,B 0,C 180,E1 -17756.444,E2 -17756.444} C_VEL
LIN {X 0,Y 270.288,Z 281.629,A -85,B 0,C 180,E1 -17760.109,E2 -17760.109} C_VEL
LIN {X 0,Y 270.205,Z 281.638,A -85,B 0,C 180,E1 -17764.905,E2 -17764.905} C_VEL
LIN {X 0,Y 270.225,Z 281.635,A -85,B 0,C 180,E1 -17768.716,E2 -17768.716} C_VEL
LIN {X 0,Y 270.17,Z 281.642,A -85,B 0,C 180,E1 -17773.249,E2 -17773.249} C_VEL
LIN {X 0,Y 270.172,Z 281.645,A -85,B 0,C 180,E1 -17777.441,E2 -17777.441} C_VEL
LIN {X 0,Y 270.208,Z 281.639,A -85,B 0,C 180,E1 -17781.373,E2 -17781.373} C_VEL
LIN {X 0,Y 270.202,Z 281.639,A -85,B 0,C 180,E1 -17785.093,E2 -17785.093} C_VEL
LIN {X 0,Y 270.201,Z 281.638,A -85,B 0,C 180,E1 -17789.129,E2 -17789.129} C_VEL
LIN {X 0,Y 270.265,Z 281.63,A -85,B 0,C 180,E1 -17792.144,E2 -17792.144} C_VEL
LIN {X 0,Y 270.277,Z 281.632,A -85,B 0,C 180,E1 -17795.518,E2 -17795.518} C_VEL
LIN {X 0,Y 270.3,Z 281.625,A -85,B 0,C 180,E1 -17800.243,E2 -17800.243} C_VEL
LIN {X 0,Y 270.395,Z 281.613,A -85,B 0,C 180,E1 -17804.934,E2 -17804.934} C_VEL
LIN {X 0,Y 270.41,Z 281.615,A -85,B 0,C 180,E1 -17809.517,E2 -17809.517} C_VEL
LIN {X 0,Y 270.596,Z 281.588,A -85,B 0,C 180,E1 -17812.537,E2 -17812.537} C_VEL
LIN {X 0,Y 270.784,Z 281.565,A -85,B 0,C 180,E1 -17818.512,E2 -17818.512} C_VEL
LIN {X 0,Y 270.783,Z 281.568,A -85,B 0,C 180,E1 -17821.486,E2 -17821.486} C_VEL
LIN {X 0,Y 270.607,Z 281.59,A -85,B 0,C 180,E1 -17827.46,E2 -17827.46} C_VEL
LIN {X 0,Y 270.438,Z 281.607,A -85,B 0,C 180,E1 -17830.48,E2 -17830.48} C_VEL
LIN {X 0,Y 270.392,Z 281.614,A -85,B 0,C 180,E1 -17835.064,E2 -17835.064} C_VEL
LIN {X 0,Y 270.298,Z 281.628,A -85,B 0,C 180,E1 -17839.754,E2 -17839.754} C_VEL
LIN {X 0,Y 270.269,Z 281.629,A -85,B 0,C 180,E1 -17844.584,E2 -17844.584} C_VEL
LIN {X 0,Y 270.264,Z 281.631,A -85,B 0,C 180,E1 -17847.908,E2 -17847.908} C_VEL
LIN {X 0,Y 270.178,Z 281.642,A -85,B 0,C 180,E1 -17851.347,E2 -17851.347} C_VEL
LIN {X 0,Y 270.218,Z 281.635,A -85,B 0,C 180,E1 -17854.901,E2 -17854.901} C_VEL
LIN {X 0,Y 270.216,Z 281.634,A -85,B 0,C 180,E1 -17858.716,E2 -17858.716} C_VEL
LIN {X 0,Y 270.195,Z 281.638,A -85,B 0,C 180,E1 -17862.551,E2 -17862.551} C_VEL
LIN {X 0,Y 270.206,Z 281.635,A -85,B 0,C 180,E1 -17866.739,E2 -17866.739} C_VEL
LIN {X 0,Y 270.239,Z 281.635,A -85,B 0,C 180,E1 -17869.446,E2 -17869.446} C_VEL
LIN {X 0,Y 270.25,Z 281.635,A -85,B 0,C 180,E1 -17873.721,E2 -17873.721} C_VEL
LIN {X 0,Y 270.197,Z 281.637,A -85,B 0,C 180,E1 -17876.892,E2 -17876.892} C_VEL
LIN {X 0,Y 270.221,Z 281.635,A -85,B 0,C 180,E1 -17880.386,E2 -17880.386} C_VEL
LIN {X 0,Y 270.256,Z 281.634,A -85,B 0,C 180,E1 -17883.763,E2 -17883.763} C_VEL
LIN {X 0,Y 270.225,Z 281.635,A -85,B 0,C 180,E1 -17887.038,E2 -17887.038} C_VEL
LIN {X 0,Y 270.294,Z 281.626,A -85,B 0,C 180,E1 -17890.244,E2 -17890.244} C_VEL
LIN {X 0,Y 270.395,Z 281.613,A -85,B 0,C 180,E1 -17894.935,E2 -17894.935} C_VEL
LIN {X 0,Y 270.434,Z 281.61,A -85,B 0,C 180,E1 -17899.519,E2 -17899.519} C_VEL
LIN {X 0,Y 270.603,Z 281.587,A -85,B 0,C 180,E1 -17902.538,E2 -17902.538} C_VEL
LIN {X 0,Y 270.779,Z 281.564,A -85,B 0,C 180,E1 -17908.512,E2 -17908.512} C_VEL
LIN {X 0,Y 270.779,Z 281.567,A -85,B 0,C 180,E1 -17911.487,E2 -17911.487} C_VEL
LIN {X 0,Y 270.599,Z 281.588,A -85,B 0,C 180,E1 -17917.461,E2 -17917.461} C_VEL
LIN {X 0,Y 270.434,Z 281.609,A -85,B 0,C 180,E1 -17920.481,E2 -17920.481} C_VEL
LIN {X 0,Y 270.395,Z 281.613,A -85,B 0,C 180,E1 -17925.064,E2 -17925.064} C_VEL
LIN {X 0,Y 270.292,Z 281.63,A -85,B 0,C 180,E1 -17929.755,E2 -17929.755} C_VEL
LIN {X 0,Y 270.229,Z 281.634,A -85,B 0,C 180,E1 -17934.589,E2 -17934.589} C_VEL
LIN {X 0,Y 270.303,Z 281.629,A -85,B 0,C 180,E1 -17938.062,E2 -17938.062} C_VEL
LIN {X 0,Y 275.639,Z 298.922,A -85,B 0,C 180,E1 -17938.923,E2 -17938.923} C_VEL
LIN {X 0,Y 276.214,Z 303.365,A -85,B 0,C 180,E1 -17939.092,E2 -17939.092} C_VEL
LIN {X 0,Y 274.779,Z 356.297,A -85,B 0,C 180,E1 -17940.707,E2 -17940.707} C_VEL
LIN {X 0,Y 274.436,Z 366.517,A -85,B 0,C 180,E1 -17941.236,E2 -17941.236} C_VEL
LIN {X 0,Y 273.777,Z 377.842,A -85,B 0,C 180,E1 -17942.103,E2 -17942.103} C_VEL
LIN {X 0,Y 273.036,Z 387.832,A -85,B 0,C 180,E1 -17943.159,E2 -17943.159} C_VEL
LIN {X 0,Y 272.383,Z 396.65,A -85,B 0,C 180,E1 -17944.348,E2 -17944.348} C_VEL
LIN {X 0,Y 271.564,Z 404.294,A -85,B 0,C 180,E1 -17945.611,E2 -17945.611} C_VEL
LIN {X 0,Y 270.639,Z 412.908,A -85,B 0,C 180,E1 -17947.372,E2 -17947.372} C_VEL
LIN {X 0,Y 269.952,Z 419.657,A -85,B 0,C 180,E1 -17949.146,E2 -17949.146} C_VEL
LIN {X 0,Y 269.336,Z 424.852,A -85,B 0,C 180,E1 -17950.827,E2 -17950.827} C_VEL
LIN {X 0,Y 268.885,Z 430.01,A -85,B 0,C 180,E1 -17952.961,E2 -17952.961} C_VEL
LIN {X 0,Y 268.471,Z 433.756,A -85,B 0,C 180,E1 -17955.027,E2 -17955.027} C_VEL
LIN {X 0,Y 268.226,Z 436.504,A -85,B 0,C 180,E1 -17957.191,E2 -17957.191} C_VEL
LIN {X 0,Y 268.222,Z 438.153,A -85,B 0,C 180,E1 -17959.45,E2 -17959.45} C_VEL
LIN {X 0,Y 268.499,Z 438.568,A -85,B 0,C 180,E1 -17961.742,E2 -17961.742} C_VEL
LIN {X 0,Y 268.736,Z 438.358,A -85,B 0,C 180,E1 -17963.025,E2 -17963.025} C_VEL
LIN {X 0,Y 269.266,Z 437.258,A -85,B 0,C 180,E1 -17964.957,E2 -17964.957} C_VEL
LIN {X 0,Y 269.936,Z 435.317,A -85,B 0,C 180,E1 -17966.857,E2 -17966.857} C_VEL
LIN {X 0,Y 270.916,Z 432.227,A -85,B 0,C 180,E1 -17968.876,E2 -17968.876} C_VEL
LIN {X 0,Y 271.819,Z 428.751,A -85,B 0,C 180,E1 -17970.579,E2 -17970.579} C_VEL
LIN {X 0,Y 273.045,Z 423.935,A -85,B 0,C 180,E1 -17972.401,E2 -17972.401} C_VEL
LIN {X 0,Y 274.476,Z 417.901,A -85,B 0,C 180,E1 -17974.198,E2 -17974.198} C_VEL
LIN {X 0,Y 276.006,Z 411.363,A -85,B 0,C 180,E1 -17975.759,E2 -17975.759} C_VEL
LIN {X 0,Y 277.341,Z 404.693,A -85,B 0,C 180,E1 -17977.071,E2 -17977.071} C_VEL
LIN {X 0,Y 278.723,Z 397.096,A -85,B 0,C 180,E1 -17978.295,E2 -17978.295} C_VEL
LIN {X 0,Y 280.327,Z 386.572,A -85,B 0,C 180,E1 -17979.645,E2 -17979.645} C_VEL
LIN {X 0,Y 281.553,Z 376.462,A -85,B 0,C 180,E1 -17980.593,E2 -17980.593} C_VEL
LIN {X 0,Y 282.395,Z 366.336,A -85,B 0,C 180,E1 -17981.303,E2 -17981.303} C_VEL
LIN {X 0,Y 282.958,Z 356.797,A -85,B 0,C 180,E1 -17981.765,E2 -17981.765} C_VEL
LIN {X 0,Y 284.825,Z 310.941,A -85,B 0,C 180,E1 -17983.189,E2 -17983.189} C_VEL
LIN {X 0,Y 279.494,Z 298.549,A -85,B 0,C 180,E1 -17984.362,E2 -17984.362} C_VEL
LIN {X 0,Y 273.35,Z 287.615,A -85,B 0,C 180,E1 -17985.674,E2 -17985.674} C_VEL
LIN {X 0,Y 272.078,Z 285.372,A -85,B 0,C 180,E1 -17985.963,E2 -17985.963} C_VEL
LIN {X 0,Y 270.642,Z 282.843,A -85,B 0,C 180,E1 -17986.294,E2 -17986.294} C_VEL
LIN {X 0,Y 270.38,Z 281.618,A -85,B 0,C 180,E1 -17986.425,E2 -17986.425} C_VEL
LIN {X 0,Y 270.54,Z 281.602,A -85,B 0,C 180,E1 -17991.034,E2 -17991.034} C_VEL
LIN {X 0,Y 270.532,Z 281.599,A -85,B 0,C 180,E1 -17994.037,E2 -17994.037} C_VEL
LIN {X 0,Y 270.448,Z 281.605,A -85,B 0,C 180,E1 -17994.831,E2 -17994.831} C_VEL
LIN {X 0,Y 269.755,Z 281.696,A -85,B 0,C 180,E1 -17996.076,E2 -17996.076} C_VEL
LIN {X 0,Y 267.024,Z 282.03,A -85,B 0,C 180,E1 -17998.111,E2 -17998.111} C_VEL
LIN {X 0,Y 264.757,Z 282.319,A -85,B 0,C 180,E1 -17999.764,E2 -17999.764} C_VEL
LIN {X 0,Y 263.811,Z 282.43,A -85,B 0,C 180,E1 -18001.041,E2 -18001.041} C_VEL
LIN {X 0,Y 263.744,Z 282.438,A -85,B 0,C 180,E1 -18001.473,E2 -18001.473} C_VEL
LIN {X 0,Y 263.566,Z 282.46,A -85,B 0,C 180,E1 -18007.663,E2 -18007.663} C_VEL
LIN {X 0,Y 263.368,Z 282.49,A -85,B 0,C 180,E1 -18010.767,E2 -18010.767} C_VEL
LIN {X 0,Y 263.34,Z 282.491,A -85,B 0,C 180,E1 -18015.48,E2 -18015.48} C_VEL
LIN {X 0,Y 263.259,Z 282.494,A -85,B 0,C 180,E1 -18020.308,E2 -18020.308} C_VEL
LIN {X 0,Y 263.206,Z 282.498,A -85,B 0,C 180,E1 -18025.293,E2 -18025.293} C_VEL
LIN {X 0,Y 263.18,Z 282.505,A -85,B 0,C 180,E1 -18028.731,E2 -18028.731} C_VEL
LIN {X 0,Y 263.131,Z 282.517,A -85,B 0,C 180,E1 -18032.29,E2 -18032.29} C_VEL
LIN {X 0,Y 263.186,Z 282.513,A -85,B 0,C 180,E1 -18035.979,E2 -18035.979} C_VEL
LIN {X 0,Y 263.138,Z 282.517,A -85,B 0,C 180,E1 -18039.868,E2 -18039.868} C_VEL
LIN {X 0,Y 263.133,Z 282.515,A -85,B 0,C 180,E1 -18043.983,E2 -18043.983} C_VEL
LIN {X 0,Y 263.124,Z 282.521,A -85,B 0,C 180,E1 -18048.408,E2 -18048.408} C_VEL
LIN {X 0,Y 263.218,Z 282.511,A -85,B 0,C 180,E1 -18053.379,E2 -18053.379} C_VEL
LIN {X 0,Y 265.336,Z 290.645,A -85,B 0,C 180,E1 -18057.115,E2 -18057.115} C_VEL
LIN {X 0,Y 267.108,Z 298.309,A -85,B 0,C 180,E1 -18060.261,E2 -18060.261} C_VEL
LIN {X 0,Y 268.178,Z 303.773,A -85,B 0,C 180,E1 -18062.301,E2 -18062.301} C_VEL
LIN {X 0,Y 270.2,Z 309.012,A -85,B 0,C 180,E1 -18062.832,E2 -18062.832} C_VEL
LIN {X 0,Y 273.953,Z 326.591,A -85,B 0,C 180,E1 -18064.063,E2 -18064.063} C_VEL
LIN {X 0,Y 276.524,Z 344.187,A -85,B 0,C 180,E1 -18065.084,E2 -18065.084} C_VEL
LIN {X 0,Y 277.372,Z 354.063,A -85,B 0,C 180,E1 -18065.56,E2 -18065.56} C_VEL
LIN {X 0,Y 275.951,Z 384.432,A -85,B 0,C 180,E1 -18066.536,E2 -18066.536} C_VEL
LIN {X 0,Y 274.9,Z 395.953,A -85,B 0,C 180,E1 -18067.133,E2 -18067.133} C_VEL
LIN {X 0,Y 273.474,Z 406.19,A -85,B 0,C 180,E1 -18067.924,E2 -18067.924} C_VEL
LIN {X 0,Y 272.051,Z 414.799,A -85,B 0,C 180,E1 -18068.798,E2 -18068.798} C_VEL
LIN {X 0,Y 270.532,Z 423.109,A -85,B 0,C 180,E1 -18069.867,E2 -18069.867} C_VEL
LIN {X 0,Y 268.892,Z 431.045,A -85,B 0,C 180,E1 -18071.129,E2 -18071.129} C_VEL
LIN {X 0,Y 267.462,Z 437.65,A -85,B 0,C 180,E1 -18072.412,E2 -18072.412} C_VEL
LIN {X 0,Y 265.877,Z 443.983,A -85,B 0,C 180,E1 -18073.887,E2 -18073.887} C_VEL
LIN {X 0,Y 264.617,Z 449.268,A -85,B 0,C 180,E1 -18075.386,E2 -18075.386} C_VEL
LIN {X 0,Y 263.606,Z 453.704,A -85,B 0,C 180,E1 -18076.903,E2 -18076.903} C_VEL
LIN {X 0,Y 262.361,Z 459.021,A -85,B 0,C 180,E1 -18079.193,E2 -18079.193} C_VEL
LIN {X 0,Y 261.64,Z 462.957,A -85,B 0,C 180,E1 -18081.505,E2 -18081.505} C_VEL
LIN {X 0,Y 261.239,Z 465.549,A -85,B 0,C 180,E1 -18083.823,E2 -18083.823} C_VEL
LIN {X 0,Y 261.167,Z 466.641,A -85,B 0,C 180,E1 -18085.37,E2 -18085.37} C_VEL
LIN {X 0,Y 261.234,Z 467.155,A -85,B 0,C 180,E1 -18086.916,E2 -18086.916} C_VEL
LIN {X 0,Y 261.261,Z 467.188,A -85,B 0,C 180,E1 -18088.459,E2 -18088.459} C_VEL
LIN {X 0,Y 261.402,Z 466.744,A -85,B 0,C 180,E1 -18090,E2 -18090} C_VEL
LIN {X 0,Y 261.308,Z 465.774,A -85,B 0,C 180,E1 -18091.542,E2 -18091.542} C_VEL
LIN {X 0,Y 261.359,Z 463.16,A -85,B 0,C 180,E1 -18093.855,E2 -18093.855} C_VEL
LIN {X 0,Y 261.399,Z 459.206,A -85,B 0,C 180,E1 -18096.174,E2 -18096.174} C_VEL
LIN {X 0,Y 261.536,Z 455.743,A -85,B 0,C 180,E1 -18097.722,E2 -18097.722} C_VEL
LIN {X 0,Y 261.875,Z 450.326,A -85,B 0,C 180,E1 -18099.656,E2 -18099.656} C_VEL
LIN {X 0,Y 262.368,Z 444.99,A -85,B 0,C 180,E1 -18101.198,E2 -18101.198} C_VEL
LIN {X 0,Y 262.976,Z 438.548,A -85,B 0,C 180,E1 -18102.737,E2 -18102.737} C_VEL
LIN {X 0,Y 264.028,Z 429.686,A -85,B 0,C 180,E1 -18104.451,E2 -18104.451} C_VEL
LIN {X 0,Y 264.948,Z 420.849,A -85,B 0,C 180,E1 -18105.777,E2 -18105.777} C_VEL
LIN {X 0,Y 265.567,Z 413.052,A -85,B 0,C 180,E1 -18106.726,E2 -18106.726} C_VEL
LIN {X 0,Y 266.56,Z 403.156,A -85,B 0,C 180,E1 -18107.65,E2 -18107.65} C_VEL
LIN {X 0,Y 267.207,Z 393.876,A -85,B 0,C 180,E1 -18108.299,E2 -18108.299} C_VEL
LIN {X 0,Y 267.581,Z 384.105,A -85,B 0,C 180,E1 -18108.776,E2 -18108.776} C_VEL
LIN {X 0,Y 268.454,Z 350.452,A -85,B 0,C 180,E1 -18109.835,E2 -18109.835} C_VEL
LIN {X 0,Y 264.231,Z 307.551,A -85,B 0,C 180,E1 -18111.468,E2 -18111.468} C_VEL
LIN {X 0,Y 265.655,Z 296.984,A -85,B 0,C 180,E1 -18115.042,E2 -18115.042} C_VEL
LIN {X 0,Y 265.066,Z 292.057,A -85,B 0,C 180,E1 -18116.791,E2 -18116.791} C_VEL
LIN {X 0,Y 263.244,Z 282.506,A -85,B 0,C 180,E1 -18120.37,E2 -18120.37} C_VEL
LIN {X 0,Y 263.154,Z 282.516,A -85,B 0,C 180,E1 -18124.114,E2 -18124.114} C_VEL
LIN {X 0,Y 263.165,Z 282.516,A -85,B 0,C 180,E1 -18127.896,E2 -18127.896} C_VEL
LIN {X 0,Y 263.131,Z 282.519,A -85,B 0,C 180,E1 -18131.891,E2 -18131.891} C_VEL
LIN {X 0,Y 263.106,Z 282.522,A -85,B 0,C 180,E1 -18136.154,E2 -18136.154} C_VEL
LIN {X 0,Y 263.106,Z 282.521,A -85,B 0,C 180,E1 -18140.126,E2 -18140.126} C_VEL
LIN {X 0,Y 263.163,Z 282.516,A -85,B 0,C 180,E1 -18144.017,E2 -18144.017} C_VEL
LIN {X 0,Y 263.133,Z 282.521,A -85,B 0,C 180,E1 -18147.711,E2 -18147.711} C_VEL
LIN {X 0,Y 263.201,Z 282.512,A -85,B 0,C 180,E1 -18151.782,E2 -18151.782} C_VEL
LIN {X 0,Y 263.226,Z 282.508,A -85,B 0,C 180,E1 -18155.199,E2 -18155.199} C_VEL
LIN {X 0,Y 263.263,Z 282.505,A -85,B 0,C 180,E1 -18159.692,E2 -18159.692} C_VEL
LIN {X 0,Y 263.343,Z 282.491,A -85,B 0,C 180,E1 -18164.52,E2 -18164.52} C_VEL
LIN {X 0,Y 263.353,Z 282.492,A -85,B 0,C 180,E1 -18169.232,E2 -18169.232} C_VEL
LIN {X 0,Y 263.556,Z 282.465,A -85,B 0,C 180,E1 -18172.337,E2 -18172.337} C_VEL
LIN {X 0,Y 263.748,Z 282.441,A -85,B 0,C 180,E1 -18178.472,E2 -18178.472} C_VEL
LIN {X 0,Y 263.748,Z 282.445,A -85,B 0,C 180,E1 -18181.526,E2 -18181.526} C_VEL
LIN {X 0,Y 263.568,Z 282.468,A -85,B 0,C 180,E1 -18187.66,E2 -18187.66} C_VEL
LIN {X 0,Y 263.37,Z 282.488,A -85,B 0,C 180,E1 -18190.764,E2 -18190.764} C_VEL
LIN {X 0,Y 263.34,Z 282.495,A -85,B 0,C 180,E1 -18195.477,E2 -18195.477} C_VEL
LIN {X 0,Y 263.264,Z 282.5,A -85,B 0,C 180,E1 -18200.305,E2 -18200.305} C_VEL
LIN {X 0,Y 263.203,Z 282.511,A -85,B 0,C 180,E1 -18205.29,E2 -18205.29} C_VEL
LIN {X 0,Y 263.17,Z 282.512,A -85,B 0,C 180,E1 -18208.729,E2 -18208.729} C_VEL
LIN {X 0,Y 263.127,Z 282.519,A -85,B 0,C 180,E1 -18212.287,E2 -18212.287} C_VEL
LIN {X 0,Y 263.186,Z 282.513,A -85,B 0,C 180,E1 -18215.976,E2 -18215.976} C_VEL
LIN {X 0,Y 263.134,Z 282.521,A -85,B 0,C 180,E1 -18219.865,E2 -18219.865} C_VEL
LIN {X 0,Y 263.137,Z 282.519,A -85,B 0,C 180,E1 -18223.979,E2 -18223.979} C_VEL
LIN {X 0,Y 263.167,Z 282.514,A -85,B 0,C 180,E1 -18228.394,E2 -18228.394} C_VEL
LIN {X 0,Y 263.182,Z 282.513,A -85,B 0,C 180,E1 -18232.107,E2 -18232.107} C_VEL
LIN {X 0,Y 263.177,Z 282.516,A -85,B 0,C 180,E1 -18235.89,E2 -18235.89} C_VEL
LIN {X 0,Y 263.144,Z 282.519,A -85,B 0,C 180,E1 -18239.506,E2 -18239.506} C_VEL
LIN {X 0,Y 263.185,Z 282.51,A -85,B 0,C 180,E1 -18243.002,E2 -18243.002} C_VEL
LIN {X 0,Y 263.176,Z 282.513,A -85,B 0,C 180,E1 -18246.386,E2 -18246.386} C_VEL
LIN {X 0,Y 263.256,Z 282.507,A -85,B 0,C 180,E1 -18249.693,E2 -18249.693} C_VEL
LIN {X 0,Y 263.343,Z 282.492,A -85,B 0,C 180,E1 -18254.522,E2 -18254.522} C_VEL
LIN {X 0,Y 263.366,Z 282.489,A -85,B 0,C 180,E1 -18259.234,E2 -18259.234} C_VEL
LIN {X 0,Y 263.565,Z 282.465,A -85,B 0,C 180,E1 -18262.338,E2 -18262.338} C_VEL
LIN {X 0,Y 263.743,Z 282.44,A -85,B 0,C 180,E1 -18268.473,E2 -18268.473} C_VEL
LIN {X 0,Y 263.743,Z 282.444,A -85,B 0,C 180,E1 -18271.527,E2 -18271.527} C_VEL
LIN {X 0,Y 263.561,Z 282.466,A -85,B 0,C 180,E1 -18277.661,E2 -18277.661} C_VEL
LIN {X 0,Y 263.366,Z 282.489,A -85,B 0,C 180,E1 -18280.765,E2 -18280.765} C_VEL
LIN {X 0,Y 263.343,Z 282.493,A -85,B 0,C 180,E1 -18285.478,E2 -18285.478} C_VEL
LIN {X 0,Y 263.254,Z 282.505,A -85,B 0,C 180,E1 -18290.307,E2 -18290.307} C_VEL
LIN {X 0,Y 263.184,Z 282.513,A -85,B 0,C 180,E1 -18295.293,E2 -18295.293} C_VEL
LIN {X 0,Y 263.277,Z 282.504,A -85,B 0,C 180,E1 -18297.681,E2 -18297.681} C_VEL
LIN {X 0,Y 269.019,Z 301.073,A -85,B 0,C 180,E1 -18298.625,E2 -18298.625} C_VEL
LIN {X 0,Y 269.304,Z 305.212,A -85,B 0,C 180,E1 -18298.774,E2 -18298.774} C_VEL
LIN {X 0,Y 267.861,Z 356.292,A -85,B 0,C 180,E1 -18300.376,E2 -18300.376} C_VEL
LIN {X 0,Y 267.514,Z 366.572,A -85,B 0,C 180,E1 -18300.916,E2 -18300.916} C_VEL
LIN {X 0,Y 266.845,Z 377.82,A -85,B 0,C 180,E1 -18301.785,E2 -18301.785} C_VEL
LIN {X 0,Y 266.119,Z 387.527,A -85,B 0,C 180,E1 -18302.824,E2 -18302.824} C_VEL
LIN {X 0,Y 265.432,Z 396.155,A -85,B 0,C 180,E1 -18303.996,E2 -18303.996} C_VEL
LIN {X 0,Y 264.669,Z 403.448,A -85,B 0,C 180,E1 -18305.203,E2 -18305.203} C_VEL
LIN {X 0,Y 263.775,Z 411.043,A -85,B 0,C 180,E1 -18306.734,E2 -18306.734} C_VEL
LIN {X 0,Y 263.05,Z 418.195,A -85,B 0,C 180,E1 -18308.515,E2 -18308.515} C_VEL
LIN {X 0,Y 262.275,Z 424.939,A -85,B 0,C 180,E1 -18310.667,E2 -18310.667} C_VEL
LIN {X 0,Y 261.824,Z 430.093,A -85,B 0,C 180,E1 -18312.828,E2 -18312.828} C_VEL
LIN {X 0,Y 261.39,Z 433.964,A -85,B 0,C 180,E1 -18314.982,E2 -18314.982} C_VEL
LIN {X 0,Y 261.181,Z 436.087,A -85,B 0,C 180,E1 -18316.595,E2 -18316.595} C_VEL
LIN {X 0,Y 261.105,Z 437.279,A -85,B 0,C 180,E1 -18317.71,E2 -18317.71} C_VEL
LIN {X 0,Y 261.15,Z 438.603,A -85,B 0,C 180,E1 -18319.77,E2 -18319.77} C_VEL
LIN {X 0,Y 261.423,Z 439.011,A -85,B 0,C 180,E1 -18321.808,E2 -18321.808} C_VEL
LIN {X 0,Y 261.854,Z 438.544,A -85,B 0,C 180,E1 -18323.812,E2 -18323.812} C_VEL
LIN {X 0,Y 262.569,Z 436.939,A -85,B 0,C 180,E1 -18326.071,E2 -18326.071} C_VEL
LIN {X 0,Y 263.622,Z 433.864,A -85,B 0,C 180,E1 -18328.548,E2 -18328.548} C_VEL
LIN {X 0,Y 265.028,Z 429.209,A -85,B 0,C 180,E1 -18331.053,E2 -18331.053} C_VEL
LIN {X 0,Y 266.338,Z 424.407,A -85,B 0,C 180,E1 -18332.925,E2 -18332.925} C_VEL
LIN {X 0,Y 267.951,Z 418.197,A -85,B 0,C 180,E1 -18334.815,E2 -18334.815} C_VEL
LIN {X 0,Y 269.359,Z 412.572,A -85,B 0,C 180,E1 -18336.202,E2 -18336.202} C_VEL
LIN {X 0,Y 270.877,Z 405.388,A -85,B 0,C 180,E1 -18337.665,E2 -18337.665} C_VEL
LIN {X 0,Y 272.215,Z 398.51,A -85,B 0,C 180,E1 -18338.812,E2 -18338.812} C_VEL
LIN {X 0,Y 273.534,Z 390.562,A -85,B 0,C 180,E1 -18339.902,E2 -18339.902} C_VEL
LIN {X 0,Y 274.623,Z 382.634,A -85,B 0,C 180,E1 -18340.782,E2 -18340.782} C_VEL
LIN {X 0,Y 275.815,Z 372.672,A -85,B 0,C 180,E1 -18341.633,E2 -18341.633} C_VEL
LIN {X 0,Y 276.675,Z 360.909,A -85,B 0,C 180,E1 -18342.349,E2 -18342.349} C_VEL
LIN {X 0,Y 277.604,Z 340.373,A -85,B 0,C 180,E1 -18343.058,E2 -18343.058} C_VEL
LIN {X 0,Y 278.754,Z 312.872,A -85,B 0,C 180,E1 -18343.927,E2 -18343.927} C_VEL
LIN {X 0,Y 274.03,Z 301.95,A -85,B 0,C 180,E1 -18345.015,E2 -18345.015} C_VEL
LIN {X 0,Y 267.639,Z 290.413,A -85,B 0,C 180,E1 -18346.471,E2 -18346.471} C_VEL
LIN {X 0,Y 265.055,Z 286.306,A -85,B 0,C 180,E1 -18347.074,E2 -18347.074} C_VEL
LIN {X 0,Y 263.57,Z 283.676,A -85,B 0,C 180,E1 -18347.44,E2 -18347.44} C_VEL
LIN {X 0,Y 263.319,Z 282.497,A -85,B 0,C 180,E1 -18347.575,E2 -18347.575} C_VEL
LIN {X 0,Y 263.465,Z 282.482,A -85,B 0,C 180,E1 -18350.791,E2 -18350.791} C_VEL
LIN {X 0,Y 263.504,Z 282.476,A -85,B 0,C 180,E1 -18353.877,E2 -18353.877} C_VEL
LIN {X 0,Y 263.745,Z 282.44,A -85,B 0,C 180,E1 -18358.474,E2 -18358.474} C_VEL
LIN {X 0,Y 263.744,Z 282.438,A -85,B 0,C 180,E1 -18361.473,E2 -18361.473} C_VEL
LIN {X 0,Y 263.098,Z 282.526,A -85,B 0,C 180,E1 -18362.745,E2 -18362.745} C_VEL
LIN {X 0,Y 260.217,Z 282.882,A -85,B 0,C 180,E1 -18364.814,E2 -18364.814} C_VEL
LIN {X 0,Y 257.725,Z 283.196,A -85,B 0,C 180,E1 -18366.498,E2 -18366.498} C_VEL
LIN {X 0,Y 256.614,Z 283.325,A -85,B 0,C 180,E1 -18367.804,E2 -18367.804} C_VEL
LIN {X 0,Y 256.503,Z 283.337,A -85,B 0,C 180,E1 -18368.248,E2 -18368.248} C_VEL
LIN {X 0,Y 256.288,Z 283.363,A -85,B 0,C 180,E1 -18372.674,E2 -18372.674} C_VEL
LIN {X 0,Y 256.257,Z 283.366,A -85,B 0,C 180,E1 -18376.287,E2 -18376.287} C_VEL
LIN {X 0,Y 256.162,Z 283.375,A -85,B 0,C 180,E1 -18380.897,E2 -18380.897} C_VEL
LIN {X 0,Y 256.186,Z 283.373,A -85,B 0,C 180,E1 -18385.14,E2 -18385.14} C_VEL
LIN {X 0,Y 256.113,Z 283.383,A -85,B 0,C 180,E1 -18389.601,E2 -18389.601} C_VEL
LIN {X 0,Y 256.083,Z 283.388,A -85,B 0,C 180,E1 -18393.292,E2 -18393.292} C_VEL
LIN {X 0,Y 256.137,Z 283.383,A -85,B 0,C 180,E1 -18397.279,E2 -18397.279} C_VEL
LIN {X 0,Y 256.084,Z 283.393,A -85,B 0,C 180,E1 -18401.199,E2 -18401.199} C_VEL
LIN {X 0,Y 256.063,Z 283.402,A -85,B 0,C 180,E1 -18405.53,E2 -18405.53} C_VEL
LIN {X 0,Y 256.054,Z 283.4,A -85,B 0,C 180,E1 -18408.798,E2 -18408.798} C_VEL
LIN {X 0,Y 256.135,Z 283.452,A -85,B 0,C 180,E1 -18412.367,E2 -18412.367} C_VEL
LIN {X 0,Y 257.813,Z 289.612,A -85,B 0,C 180,E1 -18415.339,E2 -18415.339} C_VEL
LIN {X 0,Y 259.929,Z 298.132,A -85,B 0,C 180,E1 -18419.089,E2 -18419.089} C_VEL
LIN {X 0,Y 261.005,Z 303.187,A -85,B 0,C 180,E1 -18421.084,E2 -18421.084} C_VEL
LIN {X 0,Y 264.789,Z 312.01,A -85,B 0,C 180,E1 -18422.093,E2 -18422.093} C_VEL
LIN {X 0,Y 268.355,Z 329.605,A -85,B 0,C 180,E1 -18423.366,E2 -18423.366} C_VEL
LIN {X 0,Y 270.867,Z 347.733,A -85,B 0,C 180,E1 -18424.434,E2 -18424.434} C_VEL
LIN {X 0,Y 271.328,Z 356.507,A -85,B 0,C 180,E1 -18424.833,E2 -18424.833} C_VEL
LIN {X 0,Y 269.876,Z 384.631,A -85,B 0,C 180,E1 -18425.771,E2 -18425.771} C_VEL
LIN {X 0,Y 268.617,Z 396.946,A -85,B 0,C 180,E1 -18426.463,E2 -18426.463} C_VEL
LIN {X 0,Y 267.289,Z 405.896,A -85,B 0,C 180,E1 -18427.181,E2 -18427.181} C_VEL
LIN {X 0,Y 265.791,Z 414.444,A -85,B 0,C 180,E1 -18428.07,E2 -18428.07} C_VEL
LIN {X 0,Y 264.188,Z 422.746,A -85,B 0,C 180,E1 -18429.158,E2 -18429.158} C_VEL
LIN {X 0,Y 262.473,Z 430.674,A -85,B 0,C 180,E1 -18430.446,E2 -18430.446} C_VEL
LIN {X 0,Y 260.734,Z 438.141,A -85,B 0,C 180,E1 -18431.943,E2 -18431.943} C_VEL
LIN {X 0,Y 258.709,Z 445.78,A -85,B 0,C 180,E1 -18433.833,E2 -18433.833} C_VEL
LIN {X 0,Y 257.175,Z 451.822,A -85,B 0,C 180,E1 -18435.763,E2 -18435.763} C_VEL
LIN {X 0,Y 256.214,Z 455.776,A -85,B 0,C 180,E1 -18437.324,E2 -18437.324} C_VEL
LIN {X 0,Y 255.082,Z 460.393,A -85,B 0,C 180,E1 -18439.684,E2 -18439.684} C_VEL
LIN {X 0,Y 254.406,Z 463.689,A -85,B 0,C 180,E1 -18442.061,E2 -18442.061} C_VEL
LIN {X 0,Y 254.088,Z 466.002,A -85,B 0,C 180,E1 -18444.723,E2 -18444.723} C_VEL
LIN {X 0,Y 254.141,Z 466.793,A -85,B 0,C 180,E1 -18446.83,E2 -18446.83} C_VEL
LIN {X 0,Y 254.183,Z 466.746,A -85,B 0,C 180,E1 -18448.416,E2 -18448.416} C_VEL
LIN {X 0,Y 254.317,Z 466.222,A -85,B 0,C 180,E1 -18450,E2 -18450} C_VEL
LIN {X 0,Y 254.231,Z 465.181,A -85,B 0,C 180,E1 -18451.584,E2 -18451.584} C_VEL
LIN {X 0,Y 254.294,Z 462.47,A -85,B 0,C 180,E1 -18453.962,E2 -18453.962} C_VEL
LIN {X 0,Y 254.322,Z 458.419,A -85,B 0,C 180,E1 -18456.347,E2 -18456.347} C_VEL
LIN {X 0,Y 254.615,Z 452.885,A -85,B 0,C 180,E1 -18458.732,E2 -18458.732} C_VEL
LIN {X 0,Y 255.08,Z 446.759,A -85,B 0,C 180,E1 -18460.718,E2 -18460.718} C_VEL
LIN {X 0,Y 255.67,Z 440.754,A -85,B 0,C 180,E1 -18462.3,E2 -18462.3} C_VEL
LIN {X 0,Y 256.441,Z 433.437,A -85,B 0,C 180,E1 -18463.875,E2 -18463.875} C_VEL
LIN {X 0,Y 257.183,Z 426.88,A -85,B 0,C 180,E1 -18465.047,E2 -18465.047} C_VEL
LIN {X 0,Y 257.937,Z 420.478,A -85,B 0,C 180,E1 -18466.014,E2 -18466.014} C_VEL
LIN {X 0,Y 258.582,Z 412.692,A -85,B 0,C 180,E1 -18466.988,E2 -18466.988} C_VEL
LIN {X 0,Y 259.597,Z 402.831,A -85,B 0,C 180,E1 -18467.936,E2 -18467.936} C_VEL
LIN {X 0,Y 260.259,Z 393.596,A -85,B 0,C 180,E1 -18468.601,E2 -18468.601} C_VEL
LIN {X 0,Y 260.642,Z 384.314,A -85,B 0,C 180,E1 -18469.074,E2 -18469.074} C_VEL
LIN {X 0,Y 261.505,Z 350.542,A -85,B 0,C 180,E1 -18470.18,E2 -18470.18} C_VEL
LIN {X 0,Y 257.283,Z 307.175,A -85,B 0,C 180,E1 -18471.881,E2 -18471.881} C_VEL
LIN {X 0,Y 258.636,Z 297.223,A -85,B 0,C 180,E1 -18475.339,E2 -18475.339} C_VEL
LIN {X 0,Y 257.67,Z 291.016,A -85,B 0,C 180,E1 -18477.625,E2 -18477.625} C_VEL
LIN {X 0,Y 256.175,Z 283.387,A -85,B 0,C 180,E1 -18480.557,E2 -18480.557} C_VEL
LIN {X 0,Y 256.091,Z 283.397,A -85,B 0,C 180,E1 -18485.191,E2 -18485.191} C_VEL
LIN {X 0,Y 256.125,Z 283.393,A -85,B 0,C 180,E1 -18487.272,E2 -18487.272} C_VEL
LIN {X 0,Y 256.064,Z 283.4,A -85,B 0,C 180,E1 -18491.201,E2 -18491.201} C_VEL
LIN {X 0,Y 256.046,Z 283.404,A -85,B 0,C 180,E1 -18495.532,E2 -18495.532} C_VEL
LIN {X 0,Y 256.055,Z 283.4,A -85,B 0,C 180,E1 -18498.795,E2 -18498.795} C_VEL
LIN {X 0,Y 256.131,Z 283.389,A -85,B 0,C 180,E1 -18502.866,E2 -18502.866} C_VEL
LIN {X 0,Y 256.068,Z 283.398,A -85,B 0,C 180,E1 -18506.706,E2 -18506.706} C_VEL
LIN {X 0,Y 256.114,Z 283.391,A -85,B 0,C 180,E1 -18510.399,E2 -18510.399} C_VEL
LIN {X 0,Y 256.188,Z 283.383,A -85,B 0,C 180,E1 -18514.86,E2 -18514.86} C_VEL
LIN {X 0,Y 256.166,Z 283.385,A -85,B 0,C 180,E1 -18519.104,E2 -18519.104} C_VEL
LIN {X 0,Y 256.293,Z 283.371,A -85,B 0,C 180,E1 -18524.083,E2 -18524.083} C_VEL
LIN {X 0,Y 256.291,Z 283.371,A -85,B 0,C 180,E1 -18527.326,E2 -18527.326} C_VEL
LIN {X 0,Y 256.513,Z 283.344,A -85,B 0,C 180,E1 -18532.125,E2 -18532.125} C_VEL
LIN {X 0,Y 256.496,Z 283.344,A -85,B 0,C 180,E1 -18536.857,E2 -18536.857} C_VEL
LIN {X 0,Y 256.762,Z 283.313,A -85,B 0,C 180,E1 -18539.999,E2 -18539.999} C_VEL
LIN {X 0,Y 256.496,Z 283.345,A -85,B 0,C 180,E1 -18543.14,E2 -18543.14} C_VEL
LIN {X 0,Y 256.536,Z 283.343,A -85,B 0,C 180,E1 -18547.872,E2 -18547.872} C_VEL
LIN {X 0,Y 256.306,Z 283.368,A -85,B 0,C 180,E1 -18551.065,E2 -18551.065} C_VEL
LIN {X 0,Y 256.29,Z 283.373,A -85,B 0,C 180,E1 -18555.914,E2 -18555.914} C_VEL
LIN {X 0,Y 256.213,Z 283.378,A -85,B 0,C 180,E1 -18560.889,E2 -18560.889} C_VEL
LIN {X 0,Y 256.183,Z 283.385,A -85,B 0,C 180,E1 -18565.137,E2 -18565.137} C_VEL
LIN {X 0,Y 256.105,Z 283.395,A -85,B 0,C 180,E1 -18569.599,E2 -18569.599} C_VEL
LIN {X 0,Y 256.079,Z 283.398,A -85,B 0,C 180,E1 -18573.289,E2 -18573.289} C_VEL
LIN {X 0,Y 256.135,Z 283.39,A -85,B 0,C 180,E1 -18577.277,E2 -18577.277} C_VEL
LIN {X 0,Y 256.08,Z 283.397,A -85,B 0,C 180,E1 -18581.196,E2 -18581.196} C_VEL
LIN {X 0,Y 256.071,Z 283.4,A -85,B 0,C 180,E1 -18585.525,E2 -18585.525} C_VEL
LIN {X 0,Y 256.097,Z 283.394,A -85,B 0,C 180,E1 -18588.805,E2 -18588.805} C_VEL
LIN {X 0,Y 256.148,Z 283.387,A -85,B 0,C 180,E1 -18592.871,E2 -18592.871} C_VEL
LIN {X 0,Y 256.078,Z 283.396,A -85,B 0,C 180,E1 -18596.709,E2 -18596.709} C_VEL
LIN {X 0,Y 256.131,Z 283.392,A -85,B 0,C 180,E1 -18601.404,E2 -18601.404} C_VEL
LIN {X 0,Y 256.16,Z 283.39,A -85,B 0,C 180,E1 -18605.699,E2 -18605.699} C_VEL
LIN {X 0,Y 256.159,Z 283.387,A -85,B 0,C 180,E1 -18609.104,E2 -18609.104} C_VEL
LIN {X 0,Y 256.293,Z 283.372,A -85,B 0,C 180,E1 -18614.085,E2 -18614.085} C_VEL
LIN {X 0,Y 256.302,Z 283.368,A -85,B 0,C 180,E1 -18618.934,E2 -18618.934} C_VEL
LIN {X 0,Y 256.532,Z 283.342,A -85,B 0,C 180,E1 -18622.127,E2 -18622.127} C_VEL
LIN {X 0,Y 256.706,Z 283.317,A -85,B 0,C 180,E1 -18628.431,E2 -18628.431} C_VEL
LIN {X 0,Y 256.706,Z 283.321,A -85,B 0,C 180,E1 -18631.568,E2 -18631.568} C_VEL
LIN {X 0,Y 256.529,Z 283.343,A -85,B 0,C 180,E1 -18637.873,E2 -18637.873} C_VEL
LIN {X 0,Y 256.302,Z 283.369,A -85,B 0,C 180,E1 -18641.066,E2 -18641.066} C_VEL
LIN {X 0,Y 256.292,Z 283.374,A -85,B 0,C 180,E1 -18645.915,E2 -18645.915} C_VEL
LIN {X 0,Y 256.154,Z 283.388,A -85,B 0,C 180,E1 -18650.895,E2 -18650.895} C_VEL
LIN {X 0,Y 256.163,Z 283.387,A -85,B 0,C 180,E1 -18655.13,E2 -18655.13} C_VEL
LIN {X 0,Y 256.194,Z 283.393,A -85,B 0,C 180,E1 -18657.298,E2 -18657.298} C_VEL
LIN {X 0,Y 262.164,Z 302.237,A -85,B 0,C 180,E1 -18658.287,E2 -18658.287} C_VEL
